LIN {X 0,Y 455.191,Z 1020.489,A -85,B 0,C 180,E1 17138.452,E2 17138.452} C_VEL
LIN {X 0,Y 455.669,Z 1006.442,A -85,B 0,C 180,E1 17140.566,E2 17140.566} C_VEL
LIN {X 0,Y 455.288,Z 999.068,A -85,B 0,C 180,E1 17142.573,E2 17142.573} C_VEL
LIN {X 0,Y 455.108,Z 997.219,A -85,B 0,C 180,E1 17144.205,E2 17144.205} C_VEL
LIN {X 0,Y 455.545,Z 998.35,A -85,B 0,C 180,E1 17145.874,E2 17145.874} C_VEL
LIN {X 0,Y 456.74,Z 1004.121,A -85,B 0,C 180,E1 17147.844,E2 17147.844} C_VEL
LIN {X 0,Y 457.689,Z 1016.104,A -85,B 0,C 180,E1 17149.82,E2 17149.82} C_VEL
LIN {X 0,Y 444.133,Z 1065.097,A -85,B 0,C 180,E1 17152.938,E2 17152.938} C_VEL
LIN {X 0,Y 432.896,Z 1103.693,A -85,B 0,C 180,E1 17156.355,E2 17156.355} C_VEL
LIN {X 0,Y 423.034,Z 1137.682,A -85,B 0,C 180,E1 17160.428,E2 17160.428} C_VEL
LIN {X 0,Y 415.2,Z 1166.581,A -85,B 0,C 180,E1 17165.098,E2 17165.098} C_VEL
LIN {X 0,Y 409.503,Z 1190.101,A -85,B 0,C 180,E1 17170.266,E2 17170.266} C_VEL
LIN {X 0,Y 406.234,Z 1207.399,A -85,B 0,C 180,E1 17175.641,E2 17175.641} C_VEL
LIN {X 0,Y 404.984,Z 1217.471,A -85,B 0,C 180,E1 17180.354,E2 17180.354} C_VEL
LIN {X 0,Y 404.678,Z 1223.746,A -85,B 0,C 180,E1 17185.736,E2 17185.736} C_VEL
LIN {X 0,Y 404.807,Z 1224.763,A -85,B 0,C 180,E1 17190.019,E2 17190.019} C_VEL
LIN {X 0,Y 404.778,Z 1222.047,A -85,B 0,C 180,E1 17194.3,E2 17194.3} C_VEL
LIN {X 0,Y 405.06,Z 1214.69,A -85,B 0,C 180,E1 17199.07,E2 17199.07} C_VEL
LIN {X 0,Y 406.066,Z 1201.006,A -85,B 0,C 180,E1 17204.275,E2 17204.275} C_VEL
LIN {X 0,Y 408.461,Z 1181.997,A -85,B 0,C 180,E1 17209.185,E2 17209.185} C_VEL
LIN {X 0,Y 412.41,Z 1157.442,A -85,B 0,C 180,E1 17213.787,E2 17213.787} C_VEL
LIN {X 0,Y 415.814,Z 1137.737,A -85,B 0,C 180,E1 17216.659,E2 17216.659} C_VEL
LIN {X 0,Y 414.066,Z 1125.291,A -85,B 0,C 180,E1 17218.355,E2 17218.355} C_VEL
LIN {X 0,Y 412.797,Z 1112.236,A -85,B 0,C 180,E1 17219.965,E2 17219.965} C_VEL
LIN {X 0,Y 419.177,Z 1075.451,A -85,B 0,C 180,E1 17223.278,E2 17223.278} C_VEL
LIN {X 0,Y 425.157,Z 1036.536,A -85,B 0,C 180,E1 17225.763,E2 17225.763} C_VEL
LIN {X 0,Y 427.532,Z 1011.003,A -85,B 0,C 180,E1 17226.997,E2 17226.997} C_VEL
LIN {X 0,Y 412.782,Z 969.477,A -85,B 0,C 180,E1 17229.572,E2 17229.572} C_VEL
LIN {X 0,Y 394.48,Z 923.03,A -85,B 0,C 180,E1 17232.402,E2 17232.402} C_VEL
LIN {X 0,Y 394.418,Z 923.03,A -85,B 0,C 180,E1 17239.363,E2 17239.363} C_VEL
LIN {X 0,Y 394.483,Z 923.03,A -85,B 0,C 180,E1 17244.932,E2 17244.932} C_VEL
LIN {X 0,Y 394.701,Z 923.03,A -85,B 0,C 180,E1 17251.739,E2 17251.739} C_VEL
LIN {X 0,Y 394.927,Z 923.03,A -85,B 0,C 180,E1 17257.506,E2 17257.506} C_VEL
LIN {X 0,Y 395.1,Z 923.497,A -85,B 0,C 180,E1 17261.03,E2 17261.03} C_VEL
LIN {X 0,Y 410.539,Z 954.287,A -85,B 0,C 180,E1 17264.343,E2 17264.343} C_VEL
LIN {X 0,Y 418.882,Z 977.95,A -85,B 0,C 180,E1 17266.049,E2 17266.049} C_VEL
LIN {X 0,Y 417.597,Z 1017.766,A -85,B 0,C 180,E1 17267.413,E2 17267.413} C_VEL
LIN {X 0,Y 415.215,Z 1045.588,A -85,B 0,C 180,E1 17269.12,E2 17269.12} C_VEL
LIN {X 0,Y 411.761,Z 1070.714,A -85,B 0,C 180,E1 17271.561,E2 17271.561} C_VEL
LIN {X 0,Y 407.999,Z 1092.019,A -85,B 0,C 180,E1 17274.69,E2 17274.69} C_VEL
LIN {X 0,Y 404.788,Z 1106.271,A -85,B 0,C 180,E1 17277.863,E2 17277.863} C_VEL
LIN {X 0,Y 401.89,Z 1116.644,A -85,B 0,C 180,E1 17281.618,E2 17281.618} C_VEL
LIN {X 0,Y 400.472,Z 1120.583,A -85,B 0,C 180,E1 17284.33,E2 17284.33} C_VEL
LIN {X 0,Y 399.572,Z 1121.825,A -85,B 0,C 180,E1 17286.517,E2 17286.517} C_VEL
LIN {X 0,Y 398.954,Z 1120.435,A -85,B 0,C 180,E1 17289.927,E2 17289.927} C_VEL
LIN {X 0,Y 398.958,Z 1113.006,A -85,B 0,C 180,E1 17294.154,E2 17294.154} C_VEL
LIN {X 0,Y 399.592,Z 1100.151,A -85,B 0,C 180,E1 17297.989,E2 17297.989} C_VEL
LIN {X 0,Y 400.849,Z 1081.362,A -85,B 0,C 180,E1 17301.567,E2 17301.567} C_VEL
LIN {X 0,Y 402.466,Z 1057.576,A -85,B 0,C 180,E1 17304.592,E2 17304.592} C_VEL
LIN {X 0,Y 404.027,Z 1030.386,A -85,B 0,C 180,E1 17306.89,E2 17306.89} C_VEL
LIN {X 0,Y 405.109,Z 1000.703,A -85,B 0,C 180,E1 17308.434,E2 17308.434} C_VEL
LIN {X 0,Y 404.88,Z 969.297,A -85,B 0,C 180,E1 17309.301,E2 17309.301} C_VEL
LIN {X 0,Y 394.897,Z 923.03,A -85,B 0,C 180,E1 17310.777,E2 17310.777} C_VEL
LIN {X 0,Y 394.426,Z 923.03,A -85,B 0,C 180,E1 17317.808,E2 17317.808} C_VEL
LIN {X 0,Y 394.391,Z 923.03,A -85,B 0,C 180,E1 17323.607,E2 17323.607} C_VEL
LIN {X 0,Y 394.447,Z 923.03,A -85,B 0,C 180,E1 17330.016,E2 17330.016} C_VEL
LIN {X 0,Y 394.553,Z 923.03,A -85,B 0,C 180,E1 17337.556,E2 17337.556} C_VEL
LIN {X 0,Y 394.819,Z 923.03,A -85,B 0,C 180,E1 17342.64,E2 17342.64} C_VEL
LIN {X 0,Y 395.179,Z 923.03,A -85,B 0,C 180,E1 17349.852,E2 17349.852} C_VEL
LIN {X 0,Y 395.545,Z 923.03,A -85,B 0,C 180,E1 17356.73,E2 17356.73} C_VEL
LIN {X 0,Y 396.026,Z 923.03,A -85,B 0,C 180,E1 17363.408,E2 17363.408} C_VEL
LIN {X 0,Y 396.58,Z 923.03,A -85,B 0,C 180,E1 17369.981,E2 17369.981} C_VEL
LIN {X 0,Y 395.971,Z 923.03,A -85,B 0,C 180,E1 17377.139,E2 17377.139} C_VEL
LIN {X 0,Y 395.625,Z 923.03,A -85,B 0,C 180,E1 17383.227,E2 17383.227} C_VEL
LIN {X 0,Y 395.195,Z 923.03,A -85,B 0,C 180,E1 17390.106,E2 17390.106} C_VEL
LIN {X 0,Y 394.82,Z 923.03,A -85,B 0,C 180,E1 17397.316,E2 17397.316} C_VEL
LIN {X 0,Y 394.598,Z 923.03,A -85,B 0,C 180,E1 17402.593,E2 17402.593} C_VEL
LIN {X 0,Y 394.468,Z 923.03,A -85,B 0,C 180,E1 17409.988,E2 17409.988} C_VEL
LIN {X 0,Y 394.457,Z 923.03,A -85,B 0,C 180,E1 17416.673,E2 17416.673} C_VEL
LIN {X 0,Y 394.548,Z 923.058,A -85,B 0,C 180,E1 17418.728,E2 17418.728} C_VEL
LIN {X 0,Y 410.897,Z 967.63,A -85,B 0,C 180,E1 17421.625,E2 17421.625} C_VEL
LIN {X 0,Y 422.679,Z 1006.495,A -85,B 0,C 180,E1 17424.633,E2 17424.633} C_VEL
LIN {X 0,Y 424.124,Z 1014.104,A -85,B 0,C 180,E1 17425.243,E2 17425.243} C_VEL
LIN {X 0,Y 417.97,Z 1053.429,A -85,B 0,C 180,E1 17428.199,E2 17428.199} C_VEL
LIN {X 0,Y 412.029,Z 1087.161,A -85,B 0,C 180,E1 17431.706,E2 17431.706} C_VEL
LIN {X 0,Y 406.484,Z 1116.868,A -85,B 0,C 180,E1 17435.86,E2 17435.86} C_VEL
LIN {X 0,Y 402.138,Z 1141.556,A -85,B 0,C 180,E1 17440.517,E2 17440.517} C_VEL
LIN {X 0,Y 399.018,Z 1161.589,A -85,B 0,C 180,E1 17445.747,E2 17445.747} C_VEL
LIN {X 0,Y 397.442,Z 1175.743,A -85,B 0,C 180,E1 17451.25,E2 17451.25} C_VEL
LIN {X 0,Y 396.827,Z 1183.919,A -85,B 0,C 180,E1 17456.723,E2 17456.723} C_VEL
LIN {X 0,Y 396.94,Z 1186.66,A -85,B 0,C 180,E1 17462.179,E2 17462.179} C_VEL
LIN {X 0,Y 397.795,Z 1184.171,A -85,B 0,C 180,E1 17467.638,E2 17467.638} C_VEL
LIN {X 0,Y 399.762,Z 1176.484,A -85,B 0,C 180,E1 17473.106,E2 17473.106} C_VEL
LIN {X 0,Y 403.759,Z 1163.247,A -85,B 0,C 180,E1 17478.547,E2 17478.547} C_VEL
LIN {X 0,Y 410.22,Z 1143.839,A -85,B 0,C 180,E1 17483.901,E2 17483.901} C_VEL
LIN {X 0,Y 419.067,Z 1118.652,A -85,B 0,C 180,E1 17488.832,E2 17488.832} C_VEL
LIN {X 0,Y 429.475,Z 1088.982,A -85,B 0,C 180,E1 17493.047,E2 17493.047} C_VEL
LIN {X 0,Y 442.014,Z 1052.06,A -85,B 0,C 180,E1 17496.896,E2 17496.896} C_VEL
LIN {X 0,Y 450.785,Z 1024.289,A -85,B 0,C 180,E1 17499.132,E2 17499.132} C_VEL
LIN {X 0,Y 451.859,Z 1011.926,A -85,B 0,C 180,E1 17501.112,E2 17501.112} C_VEL
LIN {X 0,Y 452.025,Z 1006.374,A -85,B 0,C 180,E1 17502.686,E2 17502.686} C_VEL
LIN {X 0,Y 452.023,Z 1004.71,A -85,B 0,C 180,E1 17504.587,E2 17504.587} C_VEL
LIN {X 0,Y 452.818,Z 1007.731,A -85,B 0,C 180,E1 17506.73,E2 17506.73} C_VEL
LIN {X 0,Y 453.398,Z 1017.576,A -85,B 0,C 180,E1 17508.786,E2 17508.786} C_VEL
LIN {X 0,Y 452.878,Z 1022.13,A -85,B 0,C 180,E1 17509.304,E2 17509.304} C_VEL
LIN {X 0,Y 439.917,Z 1063.67,A -85,B 0,C 180,E1 17511.957,E2 17511.957} C_VEL
LIN {X 0,Y 427.232,Z 1103.723,A -85,B 0,C 180,E1 17515.56,E2 17515.56} C_VEL
LIN {X 0,Y 416.484,Z 1138.178,A -85,B 0,C 180,E1 17519.798,E2 17519.798} C_VEL
LIN {X 0,Y 408.15,Z 1166.565,A -85,B 0,C 180,E1 17524.506,E2 17524.506} C_VEL
LIN {X 0,Y 402.053,Z 1189.788,A -85,B 0,C 180,E1 17529.736,E2 17529.736} C_VEL
LIN {X 0,Y 398.415,Z 1207.747,A -85,B 0,C 180,E1 17535.518,E2 17535.518} C_VEL
LIN {X 0,Y 397.016,Z 1218.96,A -85,B 0,C 180,E1 17541.263,E2 17541.263} C_VEL
LIN {X 0,Y 396.773,Z 1223.391,A -85,B 0,C 180,E1 17545.651,E2 17545.651} C_VEL
LIN {X 0,Y 396.918,Z 1224.311,A -85,B 0,C 180,E1 17550.019,E2 17550.019} C_VEL
LIN {X 0,Y 396.969,Z 1220.195,A -85,B 0,C 180,E1 17555.48,E2 17555.48} C_VEL
LIN {X 0,Y 397.36,Z 1210.042,A -85,B 0,C 180,E1 17560.98,E2 17560.98} C_VEL
LIN {X 0,Y 398.92,Z 1194.207,A -85,B 0,C 180,E1 17566.241,E2 17566.241} C_VEL
LIN {X 0,Y 402.034,Z 1172.688,A -85,B 0,C 180,E1 17571.227,E2 17571.227} C_VEL
LIN {X 0,Y 406.523,Z 1146.891,A -85,B 0,C 180,E1 17575.62,E2 17575.62} C_VEL
LIN {X 0,Y 412.088,Z 1116.105,A -85,B 0,C 180,E1 17579.539,E2 17579.539} C_VEL
LIN {X 0,Y 412.797,Z 1112.236,A -85,B 0,C 180,E1 17579.965,E2 17579.965} C_VEL
LIN {X 0,Y 411.653,Z 1098.605,A -85,B 0,C 180,E1 17581.486,E2 17581.486} C_VEL
LIN {X 0,Y 410.27,Z 1084.427,A -85,B 0,C 180,E1 17582.924,E2 17582.924} C_VEL
LIN {X 0,Y 416.384,Z 1046.661,A -85,B 0,C 180,E1 17585.619,E2 17585.619} C_VEL
LIN {X 0,Y 420.389,Z 1013.535,A -85,B 0,C 180,E1 17587.322,E2 17587.322} C_VEL
LIN {X 0,Y 406.01,Z 972.479,A -85,B 0,C 180,E1 17589.966,E2 17589.966} C_VEL
LIN {X 0,Y 386.525,Z 923.03,A -85,B 0,C 180,E1 17593.043,E2 17593.043} C_VEL
LIN {X 0,Y 386.41,Z 923.03,A -85,B 0,C 180,E1 17598.336,E2 17598.336} C_VEL
LIN {X 0,Y 386.579,Z 923.03,A -85,B 0,C 180,E1 17605.199,E2 17605.199} C_VEL
LIN {X 0,Y 386.829,Z 923.03,A -85,B 0,C 180,E1 17612.049,E2 17612.049} C_VEL
LIN {X 0,Y 387.149,Z 923.418,A -85,B 0,C 180,E1 17619.685,E2 17619.685} C_VEL
LIN {X 0,Y 390.017,Z 929.079,A -85,B 0,C 180,E1 17620.451,E2 17620.451} C_VEL
LIN {X 0,Y 403.178,Z 954.398,A -85,B 0,C 180,E1 17623.437,E2 17623.437} C_VEL
LIN {X 0,Y 412.347,Z 979.36,A -85,B 0,C 180,E1 17625.406,E2 17625.406} C_VEL
LIN {X 0,Y 411.141,Z 1018.392,A -85,B 0,C 180,E1 17626.79,E2 17626.79} C_VEL
LIN {X 0,Y 408.388,Z 1048.042,A -85,B 0,C 180,E1 17628.666,E2 17628.666} C_VEL
LIN {X 0,Y 404.74,Z 1072.75,A -85,B 0,C 180,E1 17631.143,E2 17631.143} C_VEL
LIN {X 0,Y 400.748,Z 1093.641,A -85,B 0,C 180,E1 17634.322,E2 17634.322} C_VEL
LIN {X 0,Y 397.096,Z 1108.65,A -85,B 0,C 180,E1 17637.821,E2 17637.821} C_VEL
LIN {X 0,Y 394.413,Z 1117.39,A -85,B 0,C 180,E1 17641.1,E2 17641.1} C_VEL
LIN {X 0,Y 392.608,Z 1121.967,A -85,B 0,C 180,E1 17644.417,E2 17644.417} C_VEL
LIN {X 0,Y 391.706,Z 1122.946,A -85,B 0,C 180,E1 17646.648,E2 17646.648} C_VEL
LIN {X 0,Y 391.083,Z 1121.036,A -85,B 0,C 180,E1 17650.129,E2 17650.129} C_VEL
LIN {X 0,Y 391.148,Z 1112.544,A -85,B 0,C 180,E1 17654.61,E2 17654.61} C_VEL
LIN {X 0,Y 391.797,Z 1099.582,A -85,B 0,C 180,E1 17658.321,E2 17658.321} C_VEL
LIN {X 0,Y 393.034,Z 1081.576,A -85,B 0,C 180,E1 17661.721,E2 17661.721} C_VEL
LIN {X 0,Y 394.668,Z 1057.76,A -85,B 0,C 180,E1 17664.766,E2 17664.766} C_VEL
LIN {X 0,Y 396.301,Z 1029.898,A -85,B 0,C 180,E1 17667.129,E2 17667.129} C_VEL
LIN {X 0,Y 397.389,Z 1000.153,A -85,B 0,C 180,E1 17668.672,E2 17668.672} C_VEL
LIN {X 0,Y 397.135,Z 970.302,A -85,B 0,C 180,E1 17669.506,E2 17669.506} C_VEL
LIN {X 0,Y 386.973,Z 923.03,A -85,B 0,C 180,E1 17671,E2 17671} C_VEL
LIN {X 0,Y 386.453,Z 923.03,A -85,B 0,C 180,E1 17678.731,E2 17678.731} C_VEL
LIN {X 0,Y 386.383,Z 923.03,A -85,B 0,C 180,E1 17685.232,E2 17685.232} C_VEL
LIN {X 0,Y 386.494,Z 923.03,A -85,B 0,C 180,E1 17691.443,E2 17691.443} C_VEL
LIN {X 0,Y 386.585,Z 923.03,A -85,B 0,C 180,E1 17696.802,E2 17696.802} C_VEL
LIN {X 0,Y 386.907,Z 923.03,A -85,B 0,C 180,E1 17703.939,E2 17703.939} C_VEL
LIN {X 0,Y 387.224,Z 923.03,A -85,B 0,C 180,E1 17709.491,E2 17709.491} C_VEL
LIN {X 0,Y 387.629,Z 923.03,A -85,B 0,C 180,E1 17717.063,E2 17717.063} C_VEL
LIN {X 0,Y 388.119,Z 923.03,A -85,B 0,C 180,E1 17723.273,E2 17723.273} C_VEL
LIN {X 0,Y 388.677,Z 923.03,A -85,B 0,C 180,E1 17729.98,E2 17729.98} C_VEL
LIN {X 0,Y 388.146,Z 923.03,A -85,B 0,C 180,E1 17736.687,E2 17736.687} C_VEL
LIN {X 0,Y 387.682,Z 923.03,A -85,B 0,C 180,E1 17743.503,E2 17743.503} C_VEL
LIN {X 0,Y 387.225,Z 923.03,A -85,B 0,C 180,E1 17750.539,E2 17750.539} C_VEL
LIN {X 0,Y 386.881,Z 923.03,A -85,B 0,C 180,E1 17757.925,E2 17757.925} C_VEL
LIN {X 0,Y 386.571,Z 923.03,A -85,B 0,C 180,E1 17765.87,E2 17765.87} C_VEL
LIN {X 0,Y 386.451,Z 923.03,A -85,B 0,C 180,E1 17772.014,E2 17772.014} C_VEL
LIN {X 0,Y 386.608,Z 923.177,A -85,B 0,C 180,E1 17778.099,E2 17778.099} C_VEL
LIN {X 0,Y 403.089,Z 967.84,A -85,B 0,C 180,E1 17781.079,E2 17781.079} C_VEL
LIN {X 0,Y 415.016,Z 1007.284,A -85,B 0,C 180,E1 17784.201,E2 17784.201} C_VEL
LIN {X 0,Y 416.619,Z 1016.141,A -85,B 0,C 180,E1 17784.925,E2 17784.925} C_VEL
LIN {X 0,Y 410.408,Z 1054.702,A -85,B 0,C 180,E1 17787.91,E2 17787.91} C_VEL
LIN {X 0,Y 404.319,Z 1088.358,A -85,B 0,C 180,E1 17791.492,E2 17791.492} C_VEL
LIN {X 0,Y 398.749,Z 1117.52,A -85,B 0,C 180,E1 17795.659,E2 17795.659} C_VEL
LIN {X 0,Y 394.092,Z 1143.431,A -85,B 0,C 180,E1 17800.685,E2 17800.685} C_VEL
LIN {X 0,Y 390.972,Z 1163.224,A -85,B 0,C 180,E1 17806.095,E2 17806.095} C_VEL
LIN {X 0,Y 389.616,Z 1175.758,A -85,B 0,C 180,E1 17811.073,E2 17811.073} C_VEL
LIN {X 0,Y 388.933,Z 1184.165,A -85,B 0,C 180,E1 17816.657,E2 17816.657} C_VEL
LIN {X 0,Y 389.052,Z 1187.126,A -85,B 0,C 180,E1 17822.224,E2 17822.224} C_VEL
LIN {X 0,Y 389.716,Z 1185.689,A -85,B 0,C 180,E1 17826.678,E2 17826.678} C_VEL
LIN {X 0,Y 391.543,Z 1179.288,A -85,B 0,C 180,E1 17832.253,E2 17832.253} C_VEL
LIN {X 0,Y 395.288,Z 1167.515,A -85,B 0,C 180,E1 17837.805,E2 17837.805} C_VEL
LIN {X 0,Y 401.929,Z 1148.838,A -85,B 0,C 180,E1 17843.542,E2 17843.542} C_VEL
LIN {X 0,Y 410.81,Z 1125.289,A -85,B 0,C 180,E1 17848.564,E2 17848.564} C_VEL
LIN {X 0,Y 421.943,Z 1095.977,A -85,B 0,C 180,E1 17853.1,E2 17853.1} C_VEL
LIN {X 0,Y 435.131,Z 1060.593,A -85,B 0,C 180,E1 17857.089,E2 17857.089} C_VEL
LIN {X 0,Y 446.809,Z 1027.128,A -85,B 0,C 180,E1 17859.981,E2 17859.981} C_VEL
LIN {X 0,Y 448.315,Z 1016.57,A -85,B 0,C 180,E1 17861.881,E2 17861.881} C_VEL
LIN {X 0,Y 448.619,Z 1013.196,A -85,B 0,C 180,E1 17863.088,E2 17863.088} C_VEL
LIN {X 0,Y 448.961,Z 1012.29,A -85,B 0,C 180,E1 17865.053,E2 17865.053} C_VEL
LIN {X 0,Y 449.458,Z 1015.621,A -85,B 0,C 180,E1 17866.789,E2 17866.789} C_VEL
LIN {X 0,Y 449.249,Z 1023.398,A -85,B 0,C 180,E1 17868.339,E2 17868.339} C_VEL
LIN {X 0,Y 432.879,Z 1071.725,A -85,B 0,C 180,E1 17871.686,E2 17871.686} C_VEL
LIN {X 0,Y 419.59,Z 1110.488,A -85,B 0,C 180,E1 17875.47,E2 17875.47} C_VEL
LIN {X 0,Y 408.639,Z 1143.005,A -85,B 0,C 180,E1 17879.771,E2 17879.771} C_VEL
LIN {X 0,Y 399.672,Z 1171.598,A -85,B 0,C 180,E1 17884.911,E2 17884.911} C_VEL
LIN {X 0,Y 394.089,Z 1191.813,A -85,B 0,C 180,E1 17889.835,E2 17889.835} C_VEL
LIN {X 0,Y 390.661,Z 1207.717,A -85,B 0,C 180,E1 17895.233,E2 17895.233} C_VEL
LIN {X 0,Y 389.284,Z 1217.092,A -85,B 0,C 180,E1 17899.961,E2 17899.961} C_VEL
LIN {X 0,Y 388.882,Z 1223.045,A -85,B 0,C 180,E1 17905.563,E2 17905.563} C_VEL
LIN {X 0,Y 389.032,Z 1223.821,A -85,B 0,C 180,E1 17910.02,E2 17910.02} C_VEL
LIN {X 0,Y 389.1,Z 1219.525,A -85,B 0,C 180,E1 17915.591,E2 17915.591} C_VEL
LIN {X 0,Y 389.439,Z 1210.457,A -85,B 0,C 180,E1 17920.64,E2 17920.64} C_VEL
LIN {X 0,Y 390.765,Z 1195.999,A -85,B 0,C 180,E1 17925.724,E2 17925.724} C_VEL
LIN {X 0,Y 393.948,Z 1174.002,A -85,B 0,C 180,E1 17931.095,E2 17931.095} C_VEL
LIN {X 0,Y 398.793,Z 1146.835,A -85,B 0,C 180,E1 17935.852,E2 17935.852} C_VEL
LIN {X 0,Y 404.49,Z 1116.115,A -85,B 0,C 180,E1 17939.842,E2 17939.842} C_VEL
LIN {X 0,Y 410.27,Z 1084.427,A -85,B 0,C 180,E1 17942.924,E2 17942.924} C_VEL
LIN {X 0,Y 408.992,Z 1069.918,A -85,B 0,C 180,E1 17944.271,E2 17944.271} C_VEL
LIN {X 0,Y 407.83,Z 1054.806,A -85,B 0,C 180,E1 17945.533,E2 17945.533} C_VEL
LIN {X 0,Y 412.988,Z 1015.191,A -85,B 0,C 180,E1 17947.709,E2 17947.709} C_VEL
LIN {X 0,Y 398.465,Z 973.55,A -85,B 0,C 180,E1 17950.479,E2 17950.479} C_VEL
LIN {X 0,Y 378.612,Z 923.03,A -85,B 0,C 180,E1 17953.698,E2 17953.698} C_VEL
LIN {X 0,Y 378.45,Z 923.03,A -85,B 0,C 180,E1 17960.296,E2 17960.296} C_VEL
LIN {X 0,Y 378.694,Z 923.03,A -85,B 0,C 180,E1 17966.954,E2 17966.954} C_VEL
LIN {X 0,Y 378.953,Z 923.03,A -85,B 0,C 180,E1 17973.986,E2 17973.986} C_VEL
LIN {X 0,Y 379.063,Z 923.637,A -85,B 0,C 180,E1 17978.14,E2 17978.14} C_VEL
LIN {X 0,Y 382.013,Z 929.148,A -85,B 0,C 180,E1 17979.015,E2 17979.015} C_VEL
LIN {X 0,Y 394.22,Z 951.156,A -85,B 0,C 180,E1 17982.065,E2 17982.065} C_VEL
LIN {X 0,Y 404.2,Z 975.224,A -85,B 0,C 180,E1 17984.325,E2 17984.325} C_VEL
LIN {X 0,Y 406.502,Z 984.421,A -85,B 0,C 180,E1 17984.92,E2 17984.92} C_VEL
LIN {X 0,Y 404.697,Z 1020.079,A -85,B 0,C 180,E1 17986.19,E2 17986.19} C_VEL
LIN {X 0,Y 401.963,Z 1047.836,A -85,B 0,C 180,E1 17987.96,E2 17987.96} C_VEL
LIN {X 0,Y 398.122,Z 1072.669,A -85,B 0,C 180,E1 17990.444,E2 17990.444} C_VEL
LIN {X 0,Y 393.828,Z 1093.968,A -85,B 0,C 180,E1 17993.669,E2 17993.669} C_VEL
LIN {X 0,Y 389.879,Z 1109.217,A -85,B 0,C 180,E1 17997.225,E2 17997.225} C_VEL
LIN {X 0,Y 386.636,Z 1119.204,A -85,B 0,C 180,E1 18001.122,E2 18001.122} C_VEL
LIN {X 0,Y 384.754,Z 1123.332,A -85,B 0,C 180,E1 18004.508,E2 18004.508} C_VEL
LIN {X 0,Y 383.831,Z 1123.953,A -85,B 0,C 180,E1 18006.785,E2 18006.785} C_VEL
LIN {X 0,Y 383.217,Z 1121.694,A -85,B 0,C 180,E1 18010.274,E2 18010.274} C_VEL
LIN {X 0,Y 383.241,Z 1113.809,A -85,B 0,C 180,E1 18014.407,E2 18014.407} C_VEL
LIN {X 0,Y 383.926,Z 1100.316,A -85,B 0,C 180,E1 18018.356,E2 18018.356} C_VEL
LIN {X 0,Y 385.219,Z 1081.747,A -85,B 0,C 180,E1 18021.882,E2 18021.882} C_VEL
LIN {X 0,Y 386.903,Z 1057.619,A -85,B 0,C 180,E1 18024.982,E2 18024.982} C_VEL
LIN {X 0,Y 388.555,Z 1029.791,A -85,B 0,C 180,E1 18027.344,E2 18027.344} C_VEL
LIN {X 0,Y 389.674,Z 999.259,A -85,B 0,C 180,E1 18028.914,E2 18028.914} C_VEL
LIN {X 0,Y 389.293,Z 971.002,A -85,B 0,C 180,E1 18029.716,E2 18029.716} C_VEL
LIN {X 0,Y 379.01,Z 923.03,A -85,B 0,C 180,E1 18031.312,E2 18031.312} C_VEL
LIN {X 0,Y 378.419,Z 923.03,A -85,B 0,C 180,E1 18039.714,E2 18039.714} C_VEL
LIN {X 0,Y 378.425,Z 923.03,A -85,B 0,C 180,E1 18047.225,E2 18047.225} C_VEL
LIN {X 0,Y 378.515,Z 923.03,A -85,B 0,C 180,E1 18053.193,E2 18053.193} C_VEL
LIN {X 0,Y 378.715,Z 923.03,A -85,B 0,C 180,E1 18058.734,E2 18058.734} C_VEL
LIN {X 0,Y 379.024,Z 923.03,A -85,B 0,C 180,E1 18063.969,E2 18063.969} C_VEL
LIN {X 0,Y 379.37,Z 923.03,A -85,B 0,C 180,E1 18071.399,E2 18071.399} C_VEL
LIN {X 0,Y 379.807,Z 923.03,A -85,B 0,C 180,E1 18078.506,E2 18078.506} C_VEL
LIN {X 0,Y 380.386,Z 923.03,A -85,B 0,C 180,E1 18085.423,E2 18085.423} C_VEL
LIN {X 0,Y 380.774,Z 923.03,A -85,B 0,C 180,E1 18089.98,E2 18089.98} C_VEL
LIN {X 0,Y 380.223,Z 923.03,A -85,B 0,C 180,E1 18096.827,E2 18096.827} C_VEL
LIN {X 0,Y 379.729,Z 923.03,A -85,B 0,C 180,E1 18103.792,E2 18103.792} C_VEL
LIN {X 0,Y 379.241,Z 923.03,A -85,B 0,C 180,E1 18110.991,E2 18110.991} C_VEL
LIN {X 0,Y 378.886,Z 923.03,A -85,B 0,C 180,E1 18118.663,E2 18118.663} C_VEL
LIN {X 0,Y 378.71,Z 923.03,A -85,B 0,C 180,E1 18123.932,E2 18123.932} C_VEL
LIN {X 0,Y 378.489,Z 923.03,A -85,B 0,C 180,E1 18130.658,E2 18130.658} C_VEL
LIN {X 0,Y 378.607,Z 923.253,A -85,B 0,C 180,E1 18137.439,E2 18137.439} C_VEL
LIN {X 0,Y 395.119,Z 967.893,A -85,B 0,C 180,E1 18140.502,E2 18140.502} C_VEL
LIN {X 0,Y 407.37,Z 1008.192,A -85,B 0,C 180,E1 18143.776,E2 18143.776} C_VEL
LIN {X 0,Y 409.045,Z 1018.506,A -85,B 0,C 180,E1 18144.636,E2 18144.636} C_VEL
LIN {X 0,Y 402.868,Z 1055.772,A -85,B 0,C 180,E1 18147.599,E2 18147.599} C_VEL
LIN {X 0,Y 396.693,Z 1089.099,A -85,B 0,C 180,E1 18151.221,E2 18151.221} C_VEL
LIN {X 0,Y 390.713,Z 1119.827,A -85,B 0,C 180,E1 18155.734,E2 18155.734} C_VEL
LIN {X 0,Y 386.046,Z 1145.21,A -85,B 0,C 180,E1 18160.869,E2 18160.869} C_VEL
LIN {X 0,Y 383.166,Z 1163.089,A -85,B 0,C 180,E1 18165.857,E2 18165.857} C_VEL
LIN {X 0,Y 381.77,Z 1175.747,A -85,B 0,C 180,E1 18170.888,E2 18170.888} C_VEL
LIN {X 0,Y 381.04,Z 1184.401,A -85,B 0,C 180,E1 18176.587,E2 18176.587} C_VEL
LIN {X 0,Y 381.165,Z 1187.594,A -85,B 0,C 180,E1 18182.27,E2 18182.27} C_VEL
LIN {X 0,Y 381.886,Z 1186.318,A -85,B 0,C 180,E1 18186.815,E2 18186.815} C_VEL
LIN {X 0,Y 383.838,Z 1180.174,A -85,B 0,C 180,E1 18192.502,E2 18192.502} C_VEL
LIN {X 0,Y 387.84,Z 1168.714,A -85,B 0,C 180,E1 18198.159,E2 18198.159} C_VEL
LIN {X 0,Y 394.407,Z 1151.476,A -85,B 0,C 180,E1 18203.717,E2 18203.717} C_VEL
LIN {X 0,Y 404.2,Z 1127.63,A -85,B 0,C 180,E1 18209.076,E2 18209.076} C_VEL
LIN {X 0,Y 416.587,Z 1097.444,A -85,B 0,C 180,E1 18213.894,E2 18213.894} C_VEL
LIN {X 0,Y 430.972,Z 1062.064,A -85,B 0,C 180,E1 18217.978,E2 18217.978} C_VEL
LIN {X 0,Y 442.694,Z 1032.353,A -85,B 0,C 180,E1 18220.539,E2 18220.539} C_VEL
LIN {X 0,Y 444.745,Z 1022.854,A -85,B 0,C 180,E1 18222.295,E2 18222.295} C_VEL
LIN {X 0,Y 445.053,Z 1021.301,A -85,B 0,C 180,E1 18222.768,E2 18222.768} C_VEL
LIN {X 0,Y 445.399,Z 1019.471,A -85,B 0,C 180,E1 18224.594,E2 18224.594} C_VEL
LIN {X 0,Y 445.828,Z 1021.012,A -85,B 0,C 180,E1 18226.072,E2 18226.072} C_VEL
LIN {X 0,Y 445.33,Z 1027.959,A -85,B 0,C 180,E1 18227.669,E2 18227.669} C_VEL
LIN {X 0,Y 429.521,Z 1069.82,A -85,B 0,C 180,E1 18230.574,E2 18230.574} C_VEL
LIN {X 0,Y 414.912,Z 1108.73,A -85,B 0,C 180,E1 18234.385,E2 18234.385} C_VEL
LIN {X 0,Y 402.513,Z 1142.706,A -85,B 0,C 180,E1 18238.948,E2 18238.948} C_VEL
LIN {X 0,Y 393.021,Z 1170.744,A -85,B 0,C 180,E1 18244.089,E2 18244.089} C_VEL
LIN {X 0,Y 386.563,Z 1192.091,A -85,B 0,C 180,E1 18249.425,E2 18249.425} C_VEL
LIN {X 0,Y 382.88,Z 1207.71,A -85,B 0,C 180,E1 18254.926,E2 18254.926} C_VEL
LIN {X 0,Y 381.411,Z 1216.933,A -85,B 0,C 180,E1 18259.751,E2 18259.751} C_VEL
LIN {X 0,Y 380.978,Z 1222.702,A -85,B 0,C 180,E1 18265.471,E2 18265.471} C_VEL
LIN {X 0,Y 381.147,Z 1223.296,A -85,B 0,C 180,E1 18270.02,E2 18270.02} C_VEL
LIN {X 0,Y 381.225,Z 1218.81,A -85,B 0,C 180,E1 18275.707,E2 18275.707} C_VEL
LIN {X 0,Y 381.581,Z 1209.582,A -85,B 0,C 180,E1 18280.862,E2 18280.862} C_VEL
LIN {X 0,Y 383.177,Z 1193.883,A -85,B 0,C 180,E1 18286.338,E2 18286.338} C_VEL
LIN {X 0,Y 386.392,Z 1172.445,A -85,B 0,C 180,E1 18291.527,E2 18291.527} C_VEL
LIN {X 0,Y 391.087,Z 1146.73,A -85,B 0,C 180,E1 18296.092,E2 18296.092} C_VEL
LIN {X 0,Y 396.894,Z 1116.042,A -85,B 0,C 180,E1 18300.157,E2 18300.157} C_VEL
LIN {X 0,Y 403.386,Z 1081.275,A -85,B 0,C 180,E1 18303.561,E2 18303.561} C_VEL
LIN {X 0,Y 407.83,Z 1054.806,A -85,B 0,C 180,E1 18305.533,E2 18305.533} C_VEL
LIN {X 0,Y 406.677,Z 1039.372,A -85,B 0,C 180,E1 18306.694,E2 18306.694} C_VEL
LIN {X 0,Y 405.245,Z 1023.527,A -85,B 0,C 180,E1 18307.743,E2 18307.743} C_VEL
LIN {X 0,Y 405.117,Z 1015.102,A -85,B 0,C 180,E1 18308.224,E2 18308.224} C_VEL
LIN {X 0,Y 390.195,Z 972.493,A -85,B 0,C 180,E1 18311.132,E2 18311.132} C_VEL
LIN {X 0,Y 370.613,Z 923.03,A -85,B 0,C 180,E1 18314.385,E2 18314.385} C_VEL
LIN {X 0,Y 370.519,Z 923.03,A -85,B 0,C 180,E1 18322.287,E2 18322.287} C_VEL
LIN {X 0,Y 370.801,Z 923.03,A -85,B 0,C 180,E1 18328.879,E2 18328.879} C_VEL
LIN {X 0,Y 371.103,Z 923.295,A -85,B 0,C 180,E1 18336.336,E2 18336.336} C_VEL
LIN {X 0,Y 373.684,Z 928.831,A -85,B 0,C 180,E1 18337.272,E2 18337.272} C_VEL
LIN {X 0,Y 383.739,Z 945.345,A -85,B 0,C 180,E1 18340.127,E2 18340.127} C_VEL
LIN {X 0,Y 394.853,Z 968.703,A -85,B 0,C 180,E1 18342.864,E2 18342.864} C_VEL
LIN {X 0,Y 400.37,Z 986.047,A -85,B 0,C 180,E1 18344.245,E2 18344.245} C_VEL
LIN {X 0,Y 398.413,Z 1021.249,A -85,B 0,C 180,E1 18345.534,E2 18345.534} C_VEL
LIN {X 0,Y 395.282,Z 1050.433,A -85,B 0,C 180,E1 18347.455,E2 18347.455} C_VEL
LIN {X 0,Y 391.204,Z 1074.867,A -85,B 0,C 180,E1 18349.992,E2 18349.992} C_VEL
LIN {X 0,Y 386.643,Z 1095.773,A -85,B 0,C 180,E1 18353.269,E2 18353.269} C_VEL
LIN {X 0,Y 382.739,Z 1109.854,A -85,B 0,C 180,E1 18356.607,E2 18356.607} C_VEL
LIN {X 0,Y 379.227,Z 1119.985,A -85,B 0,C 180,E1 18360.558,E2 18360.558} C_VEL
LIN {X 0,Y 376.878,Z 1124.614,A -85,B 0,C 180,E1 18364.602,E2 18364.602} C_VEL
LIN {X 0,Y 375.951,Z 1124.946,A -85,B 0,C 180,E1 18366.928,E2 18366.928} C_VEL
LIN {X 0,Y 375.339,Z 1122.238,A -85,B 0,C 180,E1 18370.44,E2 18370.44} C_VEL
LIN {X 0,Y 375.47,Z 1113.039,A -85,B 0,C 180,E1 18374.949,E2 18374.949} C_VEL
LIN {X 0,Y 376.247,Z 1098.406,A -85,B 0,C 180,E1 18378.973,E2 18378.973} C_VEL
LIN {X 0,Y 377.66,Z 1078.303,A -85,B 0,C 180,E1 18382.6,E2 18382.6} C_VEL
LIN {X 0,Y 379.401,Z 1052.882,A -85,B 0,C 180,E1 18385.669,E2 18385.669} C_VEL
LIN {X 0,Y 381.051,Z 1024.434,A -85,B 0,C 180,E1 18387.906,E2 18387.906} C_VEL
LIN {X 0,Y 382.008,Z 993.537,A -85,B 0,C 180,E1 18389.33,E2 18389.33} C_VEL
LIN {X 0,Y 381.433,Z 971.443,A -85,B 0,C 180,E1 18389.936,E2 18389.936} C_VEL
LIN {X 0,Y 371.066,Z 923.03,A -85,B 0,C 180,E1 18391.643,E2 18391.643} C_VEL
LIN {X 0,Y 370.467,Z 923.03,A -85,B 0,C 180,E1 18399.17,E2 18399.17} C_VEL
LIN {X 0,Y 370.51,Z 923.03,A -85,B 0,C 180,E1 18406.082,E2 18406.082} C_VEL
LIN {X 0,Y 370.515,Z 923.03,A -85,B 0,C 180,E1 18412.262,E2 18412.262} C_VEL
LIN {X 0,Y 370.812,Z 923.03,A -85,B 0,C 180,E1 18418.85,E2 18418.85} C_VEL
LIN {X 0,Y 371.135,Z 923.03,A -85,B 0,C 180,E1 18425.954,E2 18425.954} C_VEL
LIN {X 0,Y 371.568,Z 923.03,A -85,B 0,C 180,E1 18433.441,E2 18433.441} C_VEL
LIN {X 0,Y 372.063,Z 923.03,A -85,B 0,C 180,E1 18440.631,E2 18440.631} C_VEL
LIN {X 0,Y 372.71,Z 923.03,A -85,B 0,C 180,E1 18447.656,E2 18447.656} C_VEL
LIN {X 0,Y 372.702,Z 923.03,A -85,B 0,C 180,E1 18452.303,E2 18452.303} C_VEL
LIN {X 0,Y 372.094,Z 923.03,A -85,B 0,C 180,E1 18459.327,E2 18459.327} C_VEL
LIN {X 0,Y 371.635,Z 923.03,A -85,B 0,C 180,E1 18466.513,E2 18466.513} C_VEL
LIN {X 0,Y 371.143,Z 923.03,A -85,B 0,C 180,E1 18474.001,E2 18474.001} C_VEL
LIN {X 0,Y 370.856,Z 923.03,A -85,B 0,C 180,E1 18481.161,E2 18481.161} C_VEL
LIN {X 0,Y 370.551,Z 923.03,A -85,B 0,C 180,E1 18487.682,E2 18487.682} C_VEL
LIN {X 0,Y 370.561,Z 923.03,A -85,B 0,C 180,E1 18493.853,E2 18493.853} C_VEL
LIN {X 0,Y 370.637,Z 923.03,A -85,B 0,C 180,E1 18496.744,E2 18496.744} C_VEL
LIN {X 0,Y 387.321,Z 968.02,A -85,B 0,C 180,E1 18499.928,E2 18499.928} C_VEL
LIN {X 0,Y 399.187,Z 1007.102,A -85,B 0,C 180,E1 18503.157,E2 18503.157} C_VEL
LIN {X 0,Y 401.734,Z 1019.122,A -85,B 0,C 180,E1 18504.22,E2 18504.22} C_VEL
LIN {X 0,Y 395.355,Z 1056.72,A -85,B 0,C 180,E1 18507.27,E2 18507.27} C_VEL
LIN {X 0,Y 388.974,Z 1090.278,A -85,B 0,C 180,E1 18511.001,E2 18511.001} C_VEL
LIN {X 0,Y 382.945,Z 1120.522,A -85,B 0,C 180,E1 18515.545,E2 18515.545} C_VEL
LIN {X 0,Y 378.163,Z 1145.92,A -85,B 0,C 180,E1 18520.801,E2 18520.801} C_VEL
LIN {X 0,Y 375.202,Z 1164.087,A -85,B 0,C 180,E1 18526.014,E2 18526.014} C_VEL
LIN {X 0,Y 373.71,Z 1177.299,A -85,B 0,C 180,E1 18531.553,E2 18531.553} C_VEL
LIN {X 0,Y 373.15,Z 1184.609,A -85,B 0,C 180,E1 18536.515,E2 18536.515} C_VEL
LIN {X 0,Y 373.287,Z 1188.039,A -85,B 0,C 180,E1 18542.318,E2 18542.318} C_VEL
LIN {X 0,Y 374.038,Z 1186.961,A -85,B 0,C 180,E1 18546.959,E2 18546.959} C_VEL
LIN {X 0,Y 376.125,Z 1181.093,A -85,B 0,C 180,E1 18552.763,E2 18552.763} C_VEL
LIN {X 0,Y 380.392,Z 1169.97,A -85,B 0,C 180,E1 18558.527,E2 18558.527} C_VEL
LIN {X 0,Y 387.355,Z 1153.172,A -85,B 0,C 180,E1 18564.178,E2 18564.178} C_VEL
LIN {X 0,Y 397.624,Z 1129.977,A -85,B 0,C 180,E1 18569.604,E2 18569.604} C_VEL
LIN {X 0,Y 410.643,Z 1100.911,A -85,B 0,C 180,E1 18574.453,E2 18574.453} C_VEL
LIN {X 0,Y 426.991,Z 1064.105,A -85,B 0,C 180,E1 18578.85,E2 18578.85} C_VEL
LIN {X 0,Y 439.363,Z 1035.251,A -85,B 0,C 180,E1 18581.469,E2 18581.469} C_VEL
LIN {X 0,Y 441,Z 1029.605,A -85,B 0,C 180,E1 18582.583,E2 18582.583} C_VEL
LIN {X 0,Y 441.646,Z 1027.036,A -85,B 0,C 180,E1 18584.098,E2 18584.098} C_VEL
LIN {X 0,Y 442.118,Z 1028.78,A -85,B 0,C 180,E1 18586.129,E2 18586.129} C_VEL
LIN {X 0,Y 441.255,Z 1032.859,A -85,B 0,C 180,E1 18586.92,E2 18586.92} C_VEL
LIN {X 0,Y 424.046,Z 1074.464,A -85,B 0,C 180,E1 18589.963,E2 18589.963} C_VEL
LIN {X 0,Y 408.885,Z 1111.433,A -85,B 0,C 180,E1 18593.777,E2 18593.777} C_VEL
LIN {X 0,Y 395.903,Z 1144.218,A -85,B 0,C 180,E1 18598.37,E2 18598.37} C_VEL
LIN {X 0,Y 385.897,Z 1171.554,A -85,B 0,C 180,E1 18603.574,E2 18603.574} C_VEL
LIN {X 0,Y 379.074,Z 1192.437,A -85,B 0,C 180,E1 18608.999,E2 18608.999} C_VEL
LIN {X 0,Y 375.108,Z 1207.772,A -85,B 0,C 180,E1 18614.619,E2 18614.619} C_VEL
LIN {X 0,Y 373.386,Z 1218.289,A -85,B 0,C 180,E1 18620.706,E2 18620.706} C_VEL
LIN {X 0,Y 373.074,Z 1222.365,A -85,B 0,C 180,E1 18625.374,E2 18625.374} C_VEL
LIN {X 0,Y 373.263,Z 1222.765,A -85,B 0,C 180,E1 18630.02,E2 18630.02} C_VEL
LIN {X 0,Y 373.309,Z 1219.486,A -85,B 0,C 180,E1 18634.664,E2 18634.664} C_VEL
LIN {X 0,Y 373.602,Z 1211.139,A -85,B 0,C 180,E1 18639.918,E2 18639.918} C_VEL
LIN {X 0,Y 374.77,Z 1197.392,A -85,B 0,C 180,E1 18645.231,E2 18645.231} C_VEL
LIN {X 0,Y 377.557,Z 1177.76,A -85,B 0,C 180,E1 18650.48,E2 18650.48} C_VEL
LIN {X 0,Y 382.124,Z 1152.869,A -85,B 0,C 180,E1 18655.323,E2 18655.323} C_VEL
LIN {X 0,Y 388.171,Z 1121.899,A -85,B 0,C 180,E1 18659.778,E2 18659.778} C_VEL
LIN {X 0,Y 395.106,Z 1085.95,A -85,B 0,C 180,E1 18663.535,E2 18663.535} C_VEL
LIN {X 0,Y 401.74,Z 1047.202,A -85,B 0,C 180,E1 18666.433,E2 18666.433} C_VEL
LIN {X 0,Y 405.245,Z 1023.527,A -85,B 0,C 180,E1 18667.743,E2 18667.743} C_VEL
LIN {X 0,Y 403.425,Z 1017.493,A -85,B 0,C 180,E1 18668.211,E2 18668.211} C_VEL
LIN {X 0,Y 394.267,Z 1006.08,A -85,B 0,C 180,E1 18669.42,E2 18669.42} C_VEL
LIN {X 0,Y 377.922,Z 961.291,A -85,B 0,C 180,E1 18672.466,E2 18672.466} C_VEL
LIN {X 0,Y 362.618,Z 923.03,A -85,B 0,C 180,E1 18675.131,E2 18675.131} C_VEL
LIN {X 0,Y 362.637,Z 923.03,A -85,B 0,C 180,E1 18682.374,E2 18682.374} C_VEL
LIN {X 0,Y 362.919,Z 923.03,A -85,B 0,C 180,E1 18690.026,E2 18690.026} C_VEL
LIN {X 0,Y 363.109,Z 923.801,A -85,B 0,C 180,E1 18694.21,E2 18694.21} C_VEL
LIN {X 0,Y 365.983,Z 929.122,A -85,B 0,C 180,E1 18695.401,E2 18695.401} C_VEL
LIN {X 0,Y 368.311,Z 932.775,A -85,B 0,C 180,E1 18696.241,E2 18696.241} C_VEL
LIN {X 0,Y 377.863,Z 948.154,A -85,B 0,C 180,E1 18699.185,E2 18699.185} C_VEL
LIN {X 0,Y 388.813,Z 971.031,A -85,B 0,C 180,E1 18702.092,E2 18702.092} C_VEL
LIN {X 0,Y 394.262,Z 989.025,A -85,B 0,C 180,E1 18703.578,E2 18703.578} C_VEL
LIN {X 0,Y 392.092,Z 1024.028,A -85,B 0,C 180,E1 18704.924,E2 18704.924} C_VEL
LIN {X 0,Y 388.889,Z 1051.668,A -85,B 0,C 180,E1 18706.806,E2 18706.806} C_VEL
LIN {X 0,Y 384.466,Z 1076.398,A -85,B 0,C 180,E1 18709.429,E2 18709.429} C_VEL
LIN {X 0,Y 379.871,Z 1096.187,A -85,B 0,C 180,E1 18712.574,E2 18712.574} C_VEL
LIN {X 0,Y 375.692,Z 1110.483,A -85,B 0,C 180,E1 18715.966,E2 18715.966} C_VEL
LIN {X 0,Y 371.86,Z 1120.851,A -85,B 0,C 180,E1 18720.002,E2 18720.002} C_VEL
LIN {X 0,Y 370.291,Z 1124.189,A -85,B 0,C 180,E1 18722.341,E2 18722.341} C_VEL
LIN {X 0,Y 369.019,Z 1125.889,A -85,B 0,C 180,E1 18724.7,E2 18724.7} C_VEL
LIN {X 0,Y 368.074,Z 1125.876,A -85,B 0,C 180,E1 18727.077,E2 18727.077} C_VEL
LIN {X 0,Y 367.441,Z 1121.739,A -85,B 0,C 180,E1 18731.267,E2 18731.267} C_VEL
LIN {X 0,Y 367.654,Z 1111.68,A -85,B 0,C 180,E1 18735.636,E2 18735.636} C_VEL
LIN {X 0,Y 368.559,Z 1096.369,A -85,B 0,C 180,E1 18739.594,E2 18739.594} C_VEL
LIN {X 0,Y 370.119,Z 1074.763,A -85,B 0,C 180,E1 18743.289,E2 18743.289} C_VEL
LIN {X 0,Y 371.875,Z 1049.085,A -85,B 0,C 180,E1 18746.228,E2 18746.228} C_VEL
LIN {X 0,Y 373.484,Z 1019.914,A -85,B 0,C 180,E1 18748.394,E2 18748.394} C_VEL
LIN {X 0,Y 374.367,Z 988.394,A -85,B 0,C 180,E1 18749.709,E2 18749.709} C_VEL
LIN {X 0,Y 373.476,Z 971.424,A -85,B 0,C 180,E1 18750.181,E2 18750.181} C_VEL
LIN {X 0,Y 363.103,Z 923.03,A -85,B 0,C 180,E1 18751.834,E2 18751.834} C_VEL
LIN {X 0,Y 362.566,Z 923.03,A -85,B 0,C 180,E1 18758.698,E2 18758.698} C_VEL
LIN {X 0,Y 362.563,Z 923.03,A -85,B 0,C 180,E1 18765.119,E2 18765.119} C_VEL
LIN {X 0,Y 362.633,Z 923.03,A -85,B 0,C 180,E1 18772.352,E2 18772.352} C_VEL
LIN {X 0,Y 362.944,Z 923.03,A -85,B 0,C 180,E1 18780.004,E2 18780.004} C_VEL
LIN {X 0,Y 363.295,Z 923.03,A -85,B 0,C 180,E1 18787.995,E2 18787.995} C_VEL
LIN {X 0,Y 363.748,Z 923.03,A -85,B 0,C 180,E1 18795.546,E2 18795.546} C_VEL
LIN {X 0,Y 364.33,Z 923.03,A -85,B 0,C 180,E1 18802.832,E2 18802.832} C_VEL
LIN {X 0,Y 364.975,Z 923.03,A -85,B 0,C 180,E1 18809.979,E2 18809.979} C_VEL
LIN {X 0,Y 364.355,Z 923.03,A -85,B 0,C 180,E1 18817.125,E2 18817.125} C_VEL
LIN {X 0,Y 363.815,Z 923.03,A -85,B 0,C 180,E1 18824.408,E2 18824.408} C_VEL
LIN {X 0,Y 363.29,Z 923.03,A -85,B 0,C 180,E1 18831.96,E2 18831.96} C_VEL
LIN {X 0,Y 362.952,Z 923.03,A -85,B 0,C 180,E1 18839.946,E2 18839.946} C_VEL
LIN {X 0,Y 362.66,Z 923.03,A -85,B 0,C 180,E1 18847.654,E2 18847.654} C_VEL
LIN {X 0,Y 362.617,Z 923.03,A -85,B 0,C 180,E1 18855.072,E2 18855.072} C_VEL
LIN {X 0,Y 362.713,Z 923.03,A -85,B 0,C 180,E1 18856.047,E2 18856.047} C_VEL
LIN {X 0,Y 379.834,Z 969.241,A -85,B 0,C 180,E1 18859.419,E2 18859.419} C_VEL
LIN {X 0,Y 391.99,Z 1009.713,A -85,B 0,C 180,E1 18862.869,E2 18862.869} C_VEL
LIN {X 0,Y 394.162,Z 1021.381,A -85,B 0,C 180,E1 18863.917,E2 18863.917} C_VEL
LIN {X 0,Y 387.542,Z 1059.098,A -85,B 0,C 180,E1 18867.078,E2 18867.078} C_VEL
LIN {X 0,Y 380.832,Z 1093.315,A -85,B 0,C 180,E1 18871.023,E2 18871.023} C_VEL
LIN {X 0,Y 374.696,Z 1123.349,A -85,B 0,C 180,E1 18875.762,E2 18875.762} C_VEL
LIN {X 0,Y 370.142,Z 1147.388,A -85,B 0,C 180,E1 18880.935,E2 18880.935} C_VEL
LIN {X 0,Y 367.213,Z 1165.429,A -85,B 0,C 180,E1 18886.311,E2 18886.311} C_VEL
LIN {X 0,Y 365.775,Z 1178.038,A -85,B 0,C 180,E1 18891.803,E2 18891.803} C_VEL
LIN {X 0,Y 365.3,Z 1185.879,A -85,B 0,C 180,E1 18897.627,E2 18897.627} C_VEL
LIN {X 0,Y 365.397,Z 1188.437,A -85,B 0,C 180,E1 18902.368,E2 18902.368} C_VEL
LIN {X 0,Y 366.531,Z 1186.777,A -85,B 0,C 180,E1 18908.51,E2 18908.51} C_VEL
LIN {X 0,Y 369.119,Z 1180.299,A -85,B 0,C 180,E1 18914.216,E2 18914.216} C_VEL
LIN {X 0,Y 374.876,Z 1167.012,A -85,B 0,C 180,E1 18920.65,E2 18920.65} C_VEL
LIN {X 0,Y 383.804,Z 1147.792,A -85,B 0,C 180,E1 18926.603,E2 18926.603} C_VEL
LIN {X 0,Y 395.772,Z 1122.934,A -85,B 0,C 180,E1 18931.987,E2 18931.987} C_VEL
LIN {X 0,Y 410.692,Z 1092.312,A -85,B 0,C 180,E1 18936.717,E2 18936.717} C_VEL
LIN {X 0,Y 428.785,Z 1054.911,A -85,B 0,C 180,E1 18940.854,E2 18940.854} C_VEL
LIN {X 0,Y 435.921,Z 1039.678,A -85,B 0,C 180,E1 18942.213,E2 18942.213} C_VEL
LIN {X 0,Y 437.259,Z 1036.238,A -85,B 0,C 180,E1 18942.91,E2 18942.91} C_VEL
LIN {X 0,Y 437.878,Z 1034.522,A -85,B 0,C 180,E1 18943.642,E2 18943.642} C_VEL
LIN {X 0,Y 438.47,Z 1034.859,A -85,B 0,C 180,E1 18945.669,E2 18945.669} C_VEL
LIN {X 0,Y 437.56,Z 1037.704,A -85,B 0,C 180,E1 18946.147,E2 18946.147} C_VEL
LIN {X 0,Y 418.104,Z 1080.262,A -85,B 0,C 180,E1 18949.446,E2 18949.446} C_VEL
LIN {X 0,Y 402.081,Z 1116.218,A -85,B 0,C 180,E1 18953.4,E2 18953.4} C_VEL
LIN {X 0,Y 388.112,Z 1149.052,A -85,B 0,C 180,E1 18958.317,E2 18958.317} C_VEL
LIN {X 0,Y 377.501,Z 1176.055,A -85,B 0,C 180,E1 18963.901,E2 18963.901} C_VEL
LIN {X 0,Y 370.508,Z 1196.34,A -85,B 0,C 180,E1 18969.718,E2 18969.718} C_VEL
LIN {X 0,Y 366.755,Z 1210.706,A -85,B 0,C 180,E1 18975.71,E2 18975.71} C_VEL
LIN {X 0,Y 365.353,Z 1219.387,A -85,B 0,C 180,E1 18981.699,E2 18981.699} C_VEL
LIN {X 0,Y 365.231,Z 1222.56,A -85,B 0,C 180,E1 18987.65,E2 18987.65} C_VEL
LIN {X 0,Y 365.384,Z 1220.978,A -85,B 0,C 180,E1 18992.391,E2 18992.391} C_VEL
LIN {X 0,Y 365.528,Z 1215.586,A -85,B 0,C 180,E1 18997.199,E2 18997.199} C_VEL
LIN {X 0,Y 366.137,Z 1204.762,A -85,B 0,C 180,E1 19002.534,E2 19002.534} C_VEL
LIN {X 0,Y 368.253,Z 1187.052,A -85,B 0,C 180,E1 19008.253,E2 19008.253} C_VEL
LIN {X 0,Y 372.355,Z 1163.202,A -85,B 0,C 180,E1 19013.645,E2 19013.645} C_VEL
LIN {X 0,Y 377.962,Z 1134.891,A -85,B 0,C 180,E1 19018.326,E2 19018.326} C_VEL
LIN {X 0,Y 384.597,Z 1101.914,A -85,B 0,C 180,E1 19022.356,E2 19022.356} C_VEL
LIN {X 0,Y 391.692,Z 1063.611,A -85,B 0,C 180,E1 19025.745,E2 19025.745} C_VEL
LIN {X 0,Y 398.114,Z 1022.989,A -85,B 0,C 180,E1 19028.231,E2 19028.231} C_VEL
LIN {X 0,Y 397.282,Z 1015.488,A -85,B 0,C 180,E1 19028.719,E2 19028.719} C_VEL
LIN {X 0,Y 394.267,Z 1006.08,A -85,B 0,C 180,E1 19029.42,E2 19029.42} C_VEL
LIN {X 0,Y 388.518,Z 996.029,A -85,B 0,C 180,E1 19030.323,E2 19030.323} C_VEL
LIN {X 0,Y 378.005,Z 981.924,A -85,B 0,C 180,E1 19031.709,E2 19031.709} C_VEL
LIN {X 0,Y 377.197,Z 980.089,A -85,B 0,C 180,E1 19031.849,E2 19031.849} C_VEL
LIN {X 0,Y 354.614,Z 923.03,A -85,B 0,C 180,E1 19035.876,E2 19035.876} C_VEL
LIN {X 0,Y 354.72,Z 923.03,A -85,B 0,C 180,E1 19043.391,E2 19043.391} C_VEL
LIN {X 0,Y 355.063,Z 923.607,A -85,B 0,C 180,E1 19051.418,E2 19051.418} C_VEL
LIN {X 0,Y 357.534,Z 928.743,A -85,B 0,C 180,E1 19052.807,E2 19052.807} C_VEL
LIN {X 0,Y 360.025,Z 931.591,A -85,B 0,C 180,E1 19053.853,E2 19053.853} C_VEL
LIN {X 0,Y 367.874,Z 943.897,A -85,B 0,C 180,E1 19056.822,E2 19056.822} C_VEL
LIN {X 0,Y 378.327,Z 963.076,A -85,B 0,C 180,E1 19060.015,E2 19060.015} C_VEL
LIN {X 0,Y 387.262,Z 985.81,A -85,B 0,C 180,E1 19062.477,E2 19062.477} C_VEL
LIN {X 0,Y 388.292,Z 992.169,A -85,B 0,C 180,E1 19062.881,E2 19062.881} C_VEL
LIN {X 0,Y 386.098,Z 1024.653,A -85,B 0,C 180,E1 19064.175,E2 19064.175} C_VEL
LIN {X 0,Y 382.542,Z 1053.224,A -85,B 0,C 180,E1 19066.147,E2 19066.147} C_VEL
LIN {X 0,Y 378.023,Z 1076.906,A -85,B 0,C 180,E1 19068.692,E2 19068.692} C_VEL
LIN {X 0,Y 372.793,Z 1098.157,A -85,B 0,C 180,E1 19072.14,E2 19072.14} C_VEL
LIN {X 0,Y 368.03,Z 1113.009,A -85,B 0,C 180,E1 19075.882,E2 19075.882} C_VEL
LIN {X 0,Y 364.076,Z 1122.727,A -85,B 0,C 180,E1 19080.003,E2 19080.003} C_VEL
LIN {X 0,Y 362.471,Z 1125.758,A -85,B 0,C 180,E1 19082.392,E2 19082.392} C_VEL
LIN {X 0,Y 361.139,Z 1127.065,A -85,B 0,C 180,E1 19084.803,E2 19084.803} C_VEL
LIN {X 0,Y 359.943,Z 1126.08,A -85,B 0,C 180,E1 19088.246,E2 19088.246} C_VEL
LIN {X 0,Y 359.603,Z 1119.715,A -85,B 0,C 180,E1 19092.748,E2 19092.748} C_VEL
LIN {X 0,Y 360.07,Z 1107.535,A -85,B 0,C 180,E1 19097.086,E2 19097.086} C_VEL
LIN {X 0,Y 361.271,Z 1089.324,A -85,B 0,C 180,E1 19101.15,E2 19101.15} C_VEL
LIN {X 0,Y 362.961,Z 1066.087,A -85,B 0,C 180,E1 19104.606,E2 19104.606} C_VEL
LIN {X 0,Y 364.751,Z 1038.246,A -85,B 0,C 180,E1 19107.36,E2 19107.36} C_VEL
LIN {X 0,Y 366.088,Z 1008.706,A -85,B 0,C 180,E1 19109.185,E2 19109.185} C_VEL
LIN {X 0,Y 366.104,Z 974.325,A -85,B 0,C 180,E1 19110.322,E2 19110.322} C_VEL
LIN {X 0,Y 355.121,Z 923.03,A -85,B 0,C 180,E1 19112.195,E2 19112.195} C_VEL
LIN {X 0,Y 354.569,Z 923.03,A -85,B 0,C 180,E1 19119.877,E2 19119.877} C_VEL
LIN {X 0,Y 354.552,Z 923.03,A -85,B 0,C 180,E1 19126.982,E2 19126.982} C_VEL
LIN {X 0,Y 354.707,Z 923.03,A -85,B 0,C 180,E1 19134.044,E2 19134.044} C_VEL
LIN {X 0,Y 355.107,Z 923.03,A -85,B 0,C 180,E1 19142.068,E2 19142.068} C_VEL
LIN {X 0,Y 355.48,Z 923.03,A -85,B 0,C 180,E1 19150.098,E2 19150.098} C_VEL
LIN {X 0,Y 355.989,Z 923.03,A -85,B 0,C 180,E1 19157.726,E2 19157.726} C_VEL
LIN {X 0,Y 356.65,Z 923.03,A -85,B 0,C 180,E1 19165.118,E2 19165.118} C_VEL
LIN {X 0,Y 357.071,Z 923.03,A -85,B 0,C 180,E1 19169.979,E2 19169.979} C_VEL
LIN {X 0,Y 356.419,Z 923.03,A -85,B 0,C 180,E1 19177.285,E2 19177.285} C_VEL
LIN {X 0,Y 355.868,Z 923.03,A -85,B 0,C 180,E1 19184.737,E2 19184.737} C_VEL
LIN {X 0,Y 355.337,Z 923.03,A -85,B 0,C 180,E1 19192.478,E2 19192.478} C_VEL
LIN {X 0,Y 355.088,Z 923.03,A -85,B 0,C 180,E1 19197.885,E2 19197.885} C_VEL
LIN {X 0,Y 354.758,Z 923.03,A -85,B 0,C 180,E1 19205.967,E2 19205.967} C_VEL
LIN {X 0,Y 354.598,Z 923.03,A -85,B 0,C 180,E1 19213.574,E2 19213.574} C_VEL
LIN {X 0,Y 354.793,Z 923.792,A -85,B 0,C 180,E1 19215.374,E2 19215.374} C_VEL
LIN {X 0,Y 371.731,Z 968.77,A -85,B 0,C 180,E1 19218.762,E2 19218.762} C_VEL
LIN {X 0,Y 383.791,Z 1008.47,A -85,B 0,C 180,E1 19222.214,E2 19222.214} C_VEL
LIN {X 0,Y 386.691,Z 1023.075,A -85,B 0,C 180,E1 19223.565,E2 19223.565} C_VEL
LIN {X 0,Y 379.958,Z 1060.395,A -85,B 0,C 180,E1 19226.778,E2 19226.778} C_VEL
LIN {X 0,Y 372.911,Z 1095.136,A -85,B 0,C 180,E1 19230.902,E2 19230.902} C_VEL
LIN {X 0,Y 366.785,Z 1124.464,A -85,B 0,C 180,E1 19235.668,E2 19235.668} C_VEL
LIN {X 0,Y 362.282,Z 1147.849,A -85,B 0,C 180,E1 19240.821,E2 19240.821} C_VEL
LIN {X 0,Y 359.435,Z 1165.059,A -85,B 0,C 180,E1 19246.008,E2 19246.008} C_VEL
LIN {X 0,Y 357.924,Z 1177.76,A -85,B 0,C 180,E1 19251.5,E2 19251.5} C_VEL
LIN {X 0,Y 357.427,Z 1186.091,A -85,B 0,C 180,E1 19257.574,E2 19257.574} C_VEL
LIN {X 0,Y 357.522,Z 1188.833,A -85,B 0,C 180,E1 19262.42,E2 19262.42} C_VEL
LIN {X 0,Y 358.379,Z 1188.282,A -85,B 0,C 180,E1 19267.264,E2 19267.264} C_VEL
LIN {X 0,Y 360.75,Z 1183.02,A -85,B 0,C 180,E1 19273.317,E2 19273.317} C_VEL
LIN {X 0,Y 366.234,Z 1171.249,A -85,B 0,C 180,E1 19279.898,E2 19279.898} C_VEL
LIN {X 0,Y 374.376,Z 1154.876,A -85,B 0,C 180,E1 19285.713,E2 19285.713} C_VEL
LIN {X 0,Y 386.053,Z 1132.472,A -85,B 0,C 180,E1 19291.238,E2 19291.238} C_VEL
LIN {X 0,Y 401.524,Z 1103.32,A -85,B 0,C 180,E1 19296.349,E2 19296.349} C_VEL
LIN {X 0,Y 420.574,Z 1067.45,A -85,B 0,C 180,E1 19300.801,E2 19300.801} C_VEL
LIN {X 0,Y 433.123,Z 1043.477,A -85,B 0,C 180,E1 19303.127,E2 19303.127} C_VEL
LIN {X 0,Y 434.119,Z 1041.331,A -85,B 0,C 180,E1 19304.117,E2 19304.117} C_VEL
LIN {X 0,Y 434.493,Z 1041.562,A -85,B 0,C 180,E1 19305.274,E2 19305.274} C_VEL
LIN {X 0,Y 412.782,Z 1085.044,A -85,B 0,C 180,E1 19308.81,E2 19308.81} C_VEL
LIN {X 0,Y 395.079,Z 1121.346,A -85,B 0,C 180,E1 19313.054,E2 19313.054} C_VEL
LIN {X 0,Y 380.223,Z 1153.606,A -85,B 0,C 180,E1 19318.252,E2 19318.252} C_VEL
LIN {X 0,Y 368.979,Z 1180.514,A -85,B 0,C 180,E1 19324.281,E2 19324.281} C_VEL
LIN {X 0,Y 361.942,Z 1200.029,A -85,B 0,C 180,E1 19330.513,E2 19330.513} C_VEL
LIN {X 0,Y 358.522,Z 1212.974,A -85,B 0,C 180,E1 19336.682,E2 19336.682} C_VEL
LIN {X 0,Y 357.394,Z 1220.23,A -85,B 0,C 180,E1 19342.735,E2 19342.735} C_VEL
LIN {X 0,Y 357.364,Z 1222.087,A -85,B 0,C 180,E1 19347.598,E2 19347.598} C_VEL
LIN {X 0,Y 357.514,Z 1220.362,A -85,B 0,C 180,E1 19352.444,E2 19352.444} C_VEL
LIN {X 0,Y 357.673,Z 1213.812,A -85,B 0,C 180,E1 19357.913,E2 19357.913} C_VEL
LIN {X 0,Y 358.448,Z 1202.461,A -85,B 0,C 180,E1 19363.277,E2 19363.277} C_VEL
LIN {X 0,Y 360.622,Z 1185.604,A -85,B 0,C 180,E1 19368.654,E2 19368.654} C_VEL
LIN {X 0,Y 364.59,Z 1162.997,A -85,B 0,C 180,E1 19373.841,E2 19373.841} C_VEL
LIN {X 0,Y 370.366,Z 1134.322,A -85,B 0,C 180,E1 19378.674,E2 19378.674} C_VEL
LIN {X 0,Y 377.303,Z 1100.776,A -85,B 0,C 180,E1 19382.832,E2 19382.832} C_VEL
LIN {X 0,Y 384.509,Z 1062.685,A -85,B 0,C 180,E1 19386.236,E2 19386.236} C_VEL
LIN {X 0,Y 390.976,Z 1022.651,A -85,B 0,C 180,E1 19388.722,E2 19388.722} C_VEL
LIN {X 0,Y 379.553,Z 986.64,A -85,B 0,C 180,E1 19391.394,E2 19391.394} C_VEL
LIN {X 0,Y 377.197,Z 980.089,A -85,B 0,C 180,E1 19391.849,E2 19391.849} C_VEL
LIN {X 0,Y 368.359,Z 967.122,A -85,B 0,C 180,E1 19393.05,E2 19393.05} C_VEL
LIN {X 0,Y 359.145,Z 954.271,A -85,B 0,C 180,E1 19394.275,E2 19394.275} C_VEL
LIN {X 0,Y 346.688,Z 923.03,A -85,B 0,C 180,E1 19396.613,E2 19396.613} C_VEL
LIN {X 0,Y 346.665,Z 923.03,A -85,B 0,C 180,E1 19402.396,E2 19402.396} C_VEL
LIN {X 0,Y 346.89,Z 923.824,A -85,B 0,C 180,E1 19407.205,E2 19407.205} C_VEL
LIN {X 0,Y 350.169,Z 929.322,A -85,B 0,C 180,E1 19409.85,E2 19409.85} C_VEL
LIN {X 0,Y 352.352,Z 931.487,A -85,B 0,C 180,E1 19411.075,E2 19411.075} C_VEL
LIN {X 0,Y 357.431,Z 939.552,A -85,B 0,C 180,E1 19413.648,E2 19413.648} C_VEL
LIN {X 0,Y 364.527,Z 950.841,A -85,B 0,C 180,E1 19416.441,E2 19416.441} C_VEL
LIN {X 0,Y 373.925,Z 968.597,A -85,B 0,C 180,E1 19419.473,E2 19419.473} C_VEL
LIN {X 0,Y 382.043,Z 990.146,A -85,B 0,C 180,E1 19421.877,E2 19421.877} C_VEL
LIN {X 0,Y 382.005,Z 1001.286,A -85,B 0,C 180,E1 19422.35,E2 19422.35} C_VEL
LIN {X 0,Y 379.596,Z 1032.056,A -85,B 0,C 180,E1 19423.757,E2 19423.757} C_VEL
LIN {X 0,Y 375.481,Z 1059.307,A -85,B 0,C 180,E1 19425.881,E2 19425.881} C_VEL
LIN {X 0,Y 370.662,Z 1081.976,A -85,B 0,C 180,E1 19428.539,E2 19428.539} C_VEL
LIN {X 0,Y 365.304,Z 1101.432,A -85,B 0,C 180,E1 19431.977,E2 19431.977} C_VEL
LIN {X 0,Y 360.402,Z 1115.571,A -85,B 0,C 180,E1 19435.795,E2 19435.795} C_VEL
LIN {X 0,Y 356.283,Z 1124.573,A -85,B 0,C 180,E1 19440.003,E2 19440.003} C_VEL
LIN {X 0,Y 354.633,Z 1127.208,A -85,B 0,C 180,E1 19442.445,E2 19442.445} C_VEL
LIN {X 0,Y 353.246,Z 1128.216,A -85,B 0,C 180,E1 19444.911,E2 19444.911} C_VEL
LIN {X 0,Y 351.953,Z 1126.225,A -85,B 0,C 180,E1 19448.966,E2 19448.966} C_VEL
LIN {X 0,Y 351.73,Z 1118.264,A -85,B 0,C 180,E1 19453.67,E2 19453.67} C_VEL
LIN {X 0,Y 352.328,Z 1104.837,A -85,B 0,C 180,E1 19457.981,E2 19457.981} C_VEL
LIN {X 0,Y 353.698,Z 1085.771,A -85,B 0,C 180,E1 19461.954,E2 19461.954} C_VEL
LIN {X 0,Y 355.562,Z 1060.938,A -85,B 0,C 180,E1 19465.408,E2 19465.408} C_VEL
LIN {X 0,Y 357.366,Z 1031.907,A -85,B 0,C 180,E1 19468.05,E2 19468.05} C_VEL
LIN {X 0,Y 358.586,Z 1000.143,A -85,B 0,C 180,E1 19469.764,E2 19469.764} C_VEL
LIN {X 0,Y 358.297,Z 974.911,A -85,B 0,C 180,E1 19470.538,E2 19470.538} C_VEL
LIN {X 0,Y 347.156,Z 923.03,A -85,B 0,C 180,E1 19472.456,E2 19472.456} C_VEL
LIN {X 0,Y 346.562,Z 923.03,A -85,B 0,C 180,E1 19480.85,E2 19480.85} C_VEL
LIN {X 0,Y 346.569,Z 923.03,A -85,B 0,C 180,E1 19487.84,E2 19487.84} C_VEL
LIN {X 0,Y 346.822,Z 923.03,A -85,B 0,C 180,E1 19495.881,E2 19495.881} C_VEL
LIN {X 0,Y 347.073,Z 923.03,A -85,B 0,C 180,E1 19501.363,E2 19501.363} C_VEL
LIN {X 0,Y 347.342,Z 923.03,A -85,B 0,C 180,E1 19506.928,E2 19506.928} C_VEL
LIN {X 0,Y 347.828,Z 923.03,A -85,B 0,C 180,E1 19514.869,E2 19514.869} C_VEL
LIN {X 0,Y 348.456,Z 923.03,A -85,B 0,C 180,E1 19522.503,E2 19522.503} C_VEL
LIN {X 0,Y 349.168,Z 923.03,A -85,B 0,C 180,E1 19529.978,E2 19529.978} C_VEL
LIN {X 0,Y 348.512,Z 923.03,A -85,B 0,C 180,E1 19537.451,E2 19537.451} C_VEL
LIN {X 0,Y 347.904,Z 923.03,A -85,B 0,C 180,E1 19545.082,E2 19545.082} C_VEL
LIN {X 0,Y 347.341,Z 923.03,A -85,B 0,C 180,E1 19553.024,E2 19553.024} C_VEL
LIN {X 0,Y 347.015,Z 923.03,A -85,B 0,C 180,E1 19559.43,E2 19559.43} C_VEL
LIN {X 0,Y 346.851,Z 923.03,A -85,B 0,C 180,E1 19564.466,E2 19564.466} C_VEL
LIN {X 0,Y 346.624,Z 923.03,A -85,B 0,C 180,E1 19572.17,E2 19572.17} C_VEL
LIN {X 0,Y 346.774,Z 923.03,A -85,B 0,C 180,E1 19574.572,E2 19574.572} C_VEL
LIN {X 0,Y 364.352,Z 970.238,A -85,B 0,C 180,E1 19578.253,E2 19578.253} C_VEL
LIN {X 0,Y 376.189,Z 1009.468,A -85,B 0,C 180,E1 19581.755,E2 19581.755} C_VEL
LIN {X 0,Y 379.338,Z 1023.984,A -85,B 0,C 180,E1 19583.157,E2 19583.157} C_VEL
LIN {X 0,Y 372.287,Z 1062.084,A -85,B 0,C 180,E1 19586.518,E2 19586.518} C_VEL
LIN {X 0,Y 365.09,Z 1096.5,A -85,B 0,C 180,E1 19590.728,E2 19590.728} C_VEL
LIN {X 0,Y 359.05,Z 1124.853,A -85,B 0,C 180,E1 19595.44,E2 19595.44} C_VEL
LIN {X 0,Y 354.426,Z 1148.276,A -85,B 0,C 180,E1 19600.703,E2 19600.703} C_VEL
LIN {X 0,Y 351.405,Z 1166.347,A -85,B 0,C 180,E1 19606.317,E2 19606.317} C_VEL
LIN {X 0,Y 349.939,Z 1178.753,A -85,B 0,C 180,E1 19611.93,E2 19611.93} C_VEL
LIN {X 0,Y 349.525,Z 1186.293,A -85,B 0,C 180,E1 19617.52,E2 19617.52} C_VEL
LIN {X 0,Y 349.631,Z 1189.225,A -85,B 0,C 180,E1 19622.474,E2 19622.474} C_VEL
LIN {X 0,Y 350.657,Z 1188.735,A -85,B 0,C 180,E1 19627.831,E2 19627.831} C_VEL
LIN {X 0,Y 353.078,Z 1183.948,A -85,B 0,C 180,E1 19633.612,E2 19633.612} C_VEL
LIN {X 0,Y 358.901,Z 1172.69,A -85,B 0,C 180,E1 19640.323,E2 19640.323} C_VEL
LIN {X 0,Y 367.517,Z 1156.86,A -85,B 0,C 180,E1 19646.229,E2 19646.229} C_VEL
LIN {X 0,Y 380.456,Z 1133.994,A -85,B 0,C 180,E1 19652.086,E2 19652.086} C_VEL
LIN {X 0,Y 397.727,Z 1104.141,A -85,B 0,C 180,E1 19657.434,E2 19657.434} C_VEL
LIN {X 0,Y 418.552,Z 1068.421,A -85,B 0,C 180,E1 19661.903,E2 19661.903} C_VEL
LIN {X 0,Y 429.504,Z 1049.483,A -85,B 0,C 180,E1 19663.663,E2 19663.663} C_VEL
LIN {X 0,Y 430.371,Z 1048.293,A -85,B 0,C 180,E1 19664.603,E2 19664.603} C_VEL
LIN {X 0,Y 407.529,Z 1089.742,A -85,B 0,C 180,E1 19668.161,E2 19668.161} C_VEL
LIN {X 0,Y 389.385,Z 1123.92,A -85,B 0,C 180,E1 19672.351,E2 19672.351} C_VEL
LIN {X 0,Y 373.71,Z 1155.329,A -85,B 0,C 180,E1 19677.632,E2 19677.632} C_VEL
LIN {X 0,Y 361.862,Z 1181.304,A -85,B 0,C 180,E1 19683.737,E2 19683.737} C_VEL
LIN {X 0,Y 354.411,Z 1200.314,A -85,B 0,C 180,E1 19690.081,E2 19690.081} C_VEL
LIN {X 0,Y 350.685,Z 1213.102,A -85,B 0,C 180,E1 19696.504,E2 19696.504} C_VEL
LIN {X 0,Y 349.515,Z 1219.909,A -85,B 0,C 180,E1 19702.57,E2 19702.57} C_VEL
LIN {X 0,Y 349.467,Z 1221.608,A -85,B 0,C 180,E1 19707.544,E2 19707.544} C_VEL
LIN {X 0,Y 349.63,Z 1219.735,A -85,B 0,C 180,E1 19712.499,E2 19712.499} C_VEL
LIN {X 0,Y 349.804,Z 1212.931,A -85,B 0,C 180,E1 19718.092,E2 19718.092} C_VEL
LIN {X 0,Y 350.727,Z 1200.318,A -85,B 0,C 180,E1 19723.952,E2 19723.952} C_VEL
LIN {X 0,Y 353.307,Z 1181.904,A -85,B 0,C 180,E1 19729.662,E2 19729.662} C_VEL
LIN {X 0,Y 357.751,Z 1157.86,A -85,B 0,C 180,E1 19735.006,E2 19735.006} C_VEL
LIN {X 0,Y 364.032,Z 1127.677,A -85,B 0,C 180,E1 19739.897,E2 19739.897} C_VEL
LIN {X 0,Y 371.013,Z 1094.41,A -85,B 0,C 180,E1 19743.85,E2 19743.85} C_VEL
LIN {X 0,Y 378.029,Z 1057.607,A -85,B 0,C 180,E1 19747.041,E2 19747.041} C_VEL
LIN {X 0,Y 383.562,Z 1022.491,A -85,B 0,C 180,E1 19749.226,E2 19749.226} C_VEL
LIN {X 0,Y 369.62,Z 980.991,A -85,B 0,C 180,E1 19752.405,E2 19752.405} C_VEL
LIN {X 0,Y 359.145,Z 954.271,A -85,B 0,C 180,E1 19754.275,E2 19754.275} C_VEL
LIN {X 0,Y 352.125,Z 946.596,A -85,B 0,C 180,E1 19755.177,E2 19755.177} C_VEL
LIN {X 0,Y 344.94,Z 939.061,A -85,B 0,C 180,E1 19756.121,E2 19756.121} C_VEL
LIN {X 0,Y 342.559,Z 932.413,A -85,B 0,C 180,E1 19756.769,E2 19756.769} C_VEL
LIN {X 0,Y 342.691,Z 929.846,A -85,B 0,C 180,E1 19757.27,E2 19757.27} C_VEL
LIN {X 0,Y 342.26,Z 929.596,A -85,B 0,C 180,E1 19763.983,E2 19763.983} C_VEL
LIN {X 0,Y 344.706,Z 931.532,A -85,B 0,C 180,E1 19766.903,E2 19766.903} C_VEL
LIN {X 0,Y 348.763,Z 937.31,A -85,B 0,C 180,E1 19770.094,E2 19770.094} C_VEL
LIN {X 0,Y 354.729,Z 946.928,A -85,B 0,C 180,E1 19773.36,E2 19773.36} C_VEL
LIN {X 0,Y 363.287,Z 960.963,A -85,B 0,C 180,E1 19776.771,E2 19776.771} C_VEL
LIN {X 0,Y 372.677,Z 981.758,A -85,B 0,C 180,E1 19779.904,E2 19779.904} C_VEL
LIN {X 0,Y 376.909,Z 995.468,A -85,B 0,C 180,E1 19781.295,E2 19781.295} C_VEL
LIN {X 0,Y 374.303,Z 1027.805,A -85,B 0,C 180,E1 19782.659,E2 19782.659} C_VEL
LIN {X 0,Y 370.137,Z 1056.822,A -85,B 0,C 180,E1 19784.766,E2 19784.766} C_VEL
LIN {X 0,Y 364.675,Z 1081.434,A -85,B 0,C 180,E1 19787.593,E2 19787.593} C_VEL
LIN {X 0,Y 359.197,Z 1100.819,A -85,B 0,C 180,E1 19790.926,E2 19790.926} C_VEL
LIN {X 0,Y 353.438,Z 1116.365,A -85,B 0,C 180,E1 19795.097,E2 19795.097} C_VEL
LIN {X 0,Y 349.557,Z 1124.541,A -85,B 0,C 180,E1 19798.764,E2 19798.764} C_VEL
LIN {X 0,Y 346.789,Z 1128.647,A -85,B 0,C 180,E1 19802.5,E2 19802.5} C_VEL
LIN {X 0,Y 345.368,Z 1129.297,A -85,B 0,C 180,E1 19805.023,E2 19805.023} C_VEL
LIN {X 0,Y 344.07,Z 1126.758,A -85,B 0,C 180,E1 19809.173,E2 19809.173} C_VEL
LIN {X 0,Y 343.856,Z 1118.648,A -85,B 0,C 180,E1 19813.746,E2 19813.746} C_VEL
LIN {X 0,Y 344.422,Z 1105.836,A -85,B 0,C 180,E1 19817.888,E2 19817.888} C_VEL
LIN {X 0,Y 345.73,Z 1087.53,A -85,B 0,C 180,E1 19821.812,E2 19821.812} C_VEL
LIN {X 0,Y 347.587,Z 1063.171,A -85,B 0,C 180,E1 19825.335,E2 19825.335} C_VEL
LIN {X 0,Y 349.336,Z 1035.607,A -85,B 0,C 180,E1 19827.992,E2 19827.992} C_VEL
LIN {X 0,Y 350.716,Z 1005.777,A -85,B 0,C 180,E1 19829.767,E2 19829.767} C_VEL
LIN {X 0,Y 350.508,Z 975.871,A -85,B 0,C 180,E1 19830.751,E2 19830.751} C_VEL
LIN {X 0,Y 339.207,Z 923.03,A -85,B 0,C 180,E1 19832.757,E2 19832.757} C_VEL
LIN {X 0,Y 338.638,Z 923.03,A -85,B 0,C 180,E1 19840.632,E2 19840.632} C_VEL
LIN {X 0,Y 338.664,Z 923.03,A -85,B 0,C 180,E1 19847.962,E2 19847.962} C_VEL
LIN {X 0,Y 338.732,Z 923.03,A -85,B 0,C 180,E1 19854.53,E2 19854.53} C_VEL
LIN {X 0,Y 339.109,Z 923.03,A -85,B 0,C 180,E1 19860.626,E2 19860.626} C_VEL
LIN {X 0,Y 339.547,Z 923.03,A -85,B 0,C 180,E1 19869.122,E2 19869.122} C_VEL
LIN {X 0,Y 340.126,Z 923.03,A -85,B 0,C 180,E1 19877.144,E2 19877.144} C_VEL
LIN {X 0,Y 340.8,Z 923.03,A -85,B 0,C 180,E1 19884.89,E2 19884.89} C_VEL
LIN {X 0,Y 341.279,Z 923.03,A -85,B 0,C 180,E1 19889.978,E2 19889.978} C_VEL
LIN {X 0,Y 340.57,Z 923.03,A -85,B 0,C 180,E1 19897.626,E2 19897.626} C_VEL
LIN {X 0,Y 339.978,Z 923.03,A -85,B 0,C 180,E1 19905.442,E2 19905.442} C_VEL
LIN {X 0,Y 339.378,Z 923.03,A -85,B 0,C 180,E1 19913.597,E2 19913.597} C_VEL
LIN {X 0,Y 339.118,Z 923.03,A -85,B 0,C 180,E1 19919.322,E2 19919.322} C_VEL
LIN {X 0,Y 338.73,Z 923.03,A -85,B 0,C 180,E1 19926.579,E2 19926.579} C_VEL
LIN {X 0,Y 338.807,Z 923.03,A -85,B 0,C 180,E1 19933.825,E2 19933.825} C_VEL
LIN {X 0,Y 356.391,Z 970.001,A -85,B 0,C 180,E1 19937.581,E2 19937.581} C_VEL
LIN {X 0,Y 368.261,Z 1009.437,A -85,B 0,C 180,E1 19941.187,E2 19941.187} C_VEL
LIN {X 0,Y 371.774,Z 1026.162,A -85,B 0,C 180,E1 19942.832,E2 19942.832} C_VEL
LIN {X 0,Y 364.58,Z 1063.902,A -85,B 0,C 180,E1 19946.268,E2 19946.268} C_VEL
LIN {X 0,Y 357.269,Z 1097.809,A -85,B 0,C 180,E1 19950.545,E2 19950.545} C_VEL
LIN {X 0,Y 350.976,Z 1126.762,A -85,B 0,C 180,E1 19955.516,E2 19955.516} C_VEL
LIN {X 0,Y 346.164,Z 1151.02,A -85,B 0,C 180,E1 19961.217,E2 19961.217} C_VEL
LIN {X 0,Y 343.172,Z 1169.268,A -85,B 0,C 180,E1 19967.278,E2 19967.278} C_VEL
LIN {X 0,Y 341.828,Z 1181.739,A -85,B 0,C 180,E1 19973.629,E2 19973.629} C_VEL
LIN {X 0,Y 341.628,Z 1186.482,A -85,B 0,C 180,E1 19977.462,E2 19977.462} C_VEL
LIN {X 0,Y 341.74,Z 1189.615,A -85,B 0,C 180,E1 19982.532,E2 19982.532} C_VEL
LIN {X 0,Y 342.735,Z 1189.515,A -85,B 0,C 180,E1 19987.598,E2 19987.598} C_VEL
LIN {X 0,Y 345.416,Z 1184.894,A -85,B 0,C 180,E1 19993.92,E2 19993.92} C_VEL
LIN {X 0,Y 351.616,Z 1174.128,A -85,B 0,C 180,E1 20000.763,E2 20000.763} C_VEL
LIN {X 0,Y 361.811,Z 1157.029,A -85,B 0,C 180,E1 20007.346,E2 20007.346} C_VEL
LIN {X 0,Y 376.494,Z 1133.257,A -85,B 0,C 180,E1 20013.492,E2 20013.492} C_VEL
LIN {X 0,Y 395.205,Z 1103.695,A -85,B 0,C 180,E1 20018.761,E2 20018.761} C_VEL
LIN {X 0,Y 417.435,Z 1068.988,A -85,B 0,C 180,E1 20023.096,E2 20023.096} C_VEL
LIN {X 0,Y 423.385,Z 1059.649,A -85,B 0,C 180,E1 20023.994,E2 20023.994} C_VEL
LIN {X 0,Y 423.616,Z 1059.371,A -85,B 0,C 180,E1 20024.272,E2 20024.272} C_VEL
LIN {X 0,Y 401.238,Z 1096.499,A -85,B 0,C 180,E1 20027.717,E2 20027.717} C_VEL
LIN {X 0,Y 381.33,Z 1130.926,A -85,B 0,C 180,E1 20032.278,E2 20032.278} C_VEL
LIN {X 0,Y 364.258,Z 1162.757,A -85,B 0,C 180,E1 20038.202,E2 20038.202} C_VEL
LIN {X 0,Y 352.456,Z 1187.066,A -85,B 0,C 180,E1 20044.639,E2 20044.639} C_VEL
LIN {X 0,Y 345.833,Z 1203.561,A -85,B 0,C 180,E1 20050.895,E2 20050.895} C_VEL
LIN {X 0,Y 342.515,Z 1214.634,A -85,B 0,C 180,E1 20057.28,E2 20057.28} C_VEL
LIN {X 0,Y 341.621,Z 1219.591,A -85,B 0,C 180,E1 20062.398,E2 20062.398} C_VEL
LIN {X 0,Y 341.572,Z 1221.128,A -85,B 0,C 180,E1 20067.487,E2 20067.487} C_VEL
LIN {X 0,Y 341.749,Z 1219.081,A -85,B 0,C 180,E1 20072.556,E2 20072.556} C_VEL
LIN {X 0,Y 341.932,Z 1212.033,A -85,B 0,C 180,E1 20078.28,E2 20078.28} C_VEL
LIN {X 0,Y 342.901,Z 1199.307,A -85,B 0,C 180,E1 20084.199,E2 20084.199} C_VEL
LIN {X 0,Y 345.632,Z 1180.333,A -85,B 0,C 180,E1 20090.118,E2 20090.118} C_VEL
LIN {X 0,Y 350.363,Z 1155.812,A -85,B 0,C 180,E1 20095.571,E2 20095.571} C_VEL
LIN {X 0,Y 356.519,Z 1126.981,A -85,B 0,C 180,E1 20100.282,E2 20100.282} C_VEL
LIN {X 0,Y 363.966,Z 1092.398,A -85,B 0,C 180,E1 20104.433,E2 20104.433} C_VEL
LIN {X 0,Y 371.469,Z 1053.48,A -85,B 0,C 180,E1 20107.797,E2 20107.797} C_VEL
LIN {X 0,Y 376.304,Z 1024.941,A -85,B 0,C 180,E1 20109.57,E2 20109.57} C_VEL
LIN {X 0,Y 362.709,Z 983.953,A -85,B 0,C 180,E1 20112.825,E2 20112.825} C_VEL
LIN {X 0,Y 344.94,Z 939.061,A -85,B 0,C 180,E1 20116.121,E2 20116.121} C_VEL
LIN {X 0,Y 342.32,Z 935.82,A -85,B 0,C 180,E1 20117.032,E2 20117.032} C_VEL
LIN {X 0,Y 339.769,Z 936.833,A -85,B 0,C 180,E1 20119.973,E2 20119.973} C_VEL
LIN {X 0,Y 342.46,Z 938.454,A -85,B 0,C 180,E1 20126.399,E2 20126.399} C_VEL
LIN {X 0,Y 346.247,Z 944.599,A -85,B 0,C 180,E1 20129.713,E2 20129.713} C_VEL
LIN {X 0,Y 352.88,Z 955.508,A -85,B 0,C 180,E1 20133.447,E2 20133.447} C_VEL
LIN {X 0,Y 361.429,Z 970.912,A -85,B 0,C 180,E1 20136.938,E2 20136.938} C_VEL
LIN {X 0,Y 369.475,Z 990.676,A -85,B 0,C 180,E1 20139.753,E2 20139.753} C_VEL
LIN {X 0,Y 371.366,Z 999.088,A -85,B 0,C 180,E1 20140.517,E2 20140.517} C_VEL
LIN {X 0,Y 368.593,Z 1029.776,A -85,B 0,C 180,E1 20141.867,E2 20141.867} C_VEL
LIN {X 0,Y 364.336,Z 1057.26,A -85,B 0,C 180,E1 20143.9,E2 20143.9} C_VEL
LIN {X 0,Y 358.562,Z 1082.14,A -85,B 0,C 180,E1 20146.755,E2 20146.755} C_VEL
LIN {X 0,Y 352.718,Z 1101.538,A -85,B 0,C 180,E1 20150.135,E2 20150.135} C_VEL
LIN {X 0,Y 347.357,Z 1115.466,A -85,B 0,C 180,E1 20153.759,E2 20153.759} C_VEL
LIN {X 0,Y 342.389,Z 1125.489,A -85,B 0,C 180,E1 20158.106,E2 20158.106} C_VEL
LIN {X 0,Y 338.915,Z 1130.001,A -85,B 0,C 180,E1 20162.558,E2 20162.558} C_VEL
LIN {X 0,Y 337.463,Z 1130.291,A -85,B 0,C 180,E1 20165.141,E2 20165.141} C_VEL
LIN {X 0,Y 336.193,Z 1127.22,A -85,B 0,C 180,E1 20169.33,E2 20169.33} C_VEL
LIN {X 0,Y 335.984,Z 1118.638,A -85,B 0,C 180,E1 20173.967,E2 20173.967} C_VEL
LIN {X 0,Y 336.622,Z 1104.86,A -85,B 0,C 180,E1 20178.317,E2 20178.317} C_VEL
LIN {X 0,Y 338.039,Z 1085.43,A -85,B 0,C 180,E1 20182.335,E2 20182.335} C_VEL
LIN {X 0,Y 339.896,Z 1061.712,A -85,B 0,C 180,E1 20185.691,E2 20185.691} C_VEL
LIN {X 0,Y 341.721,Z 1032.913,A -85,B 0,C 180,E1 20188.401,E2 20188.401} C_VEL
LIN {X 0,Y 343.047,Z 1001.14,A -85,B 0,C 180,E1 20190.175,E2 20190.175} C_VEL
LIN {X 0,Y 342.556,Z 976.223,A -85,B 0,C 180,E1 20190.984,E2 20190.984} C_VEL
LIN {X 0,Y 331.271,Z 923.03,A -85,B 0,C 180,E1 20193.036,E2 20193.036} C_VEL
LIN {X 0,Y 330.709,Z 923.03,A -85,B 0,C 180,E1 20199.773,E2 20199.773} C_VEL
LIN {X 0,Y 330.71,Z 923.03,A -85,B 0,C 180,E1 20206.981,E2 20206.981} C_VEL
LIN {X 0,Y 330.777,Z 923.03,A -85,B 0,C 180,E1 20213.542,E2 20213.542} C_VEL
LIN {X 0,Y 331.119,Z 923.03,A -85,B 0,C 180,E1 20220.127,E2 20220.127} C_VEL
LIN {X 0,Y 331.552,Z 923.03,A -85,B 0,C 180,E1 20228.594,E2 20228.594} C_VEL
LIN {X 0,Y 332.16,Z 923.03,A -85,B 0,C 180,E1 20236.83,E2 20236.83} C_VEL
LIN {X 0,Y 332.886,Z 923.03,A -85,B 0,C 180,E1 20244.769,E2 20244.769} C_VEL
LIN {X 0,Y 333.375,Z 923.03,A -85,B 0,C 180,E1 20249.977,E2 20249.977} C_VEL
LIN {X 0,Y 332.63,Z 923.03,A -85,B 0,C 180,E1 20257.809,E2 20257.809} C_VEL
LIN {X 0,Y 331.997,Z 923.03,A -85,B 0,C 180,E1 20265.823,E2 20265.823} C_VEL
LIN {X 0,Y 331.602,Z 923.03,A -85,B 0,C 180,E1 20271.353,E2 20271.353} C_VEL
LIN {X 0,Y 331.135,Z 923.03,A -85,B 0,C 180,E1 20279.878,E2 20279.878} C_VEL
LIN {X 0,Y 330.852,Z 923.03,A -85,B 0,C 180,E1 20286.391,E2 20286.391} C_VEL
LIN {X 0,Y 330.814,Z 923.03,A -85,B 0,C 180,E1 20293.038,E2 20293.038} C_VEL
LIN {X 0,Y 348.415,Z 969.756,A -85,B 0,C 180,E1 20296.894,E2 20296.894} C_VEL
LIN {X 0,Y 360.296,Z 1009.157,A -85,B 0,C 180,E1 20300.577,E2 20300.577} C_VEL
LIN {X 0,Y 364.346,Z 1027.357,A -85,B 0,C 180,E1 20302.429,E2 20302.429} C_VEL
LIN {X 0,Y 356.935,Z 1065.292,A -85,B 0,C 180,E1 20305.98,E2 20305.98} C_VEL
LIN {X 0,Y 349.366,Z 1099.401,A -85,B 0,C 180,E1 20310.406,E2 20310.406} C_VEL
LIN {X 0,Y 343.228,Z 1127.051,A -85,B 0,C 180,E1 20315.273,E2 20315.273} C_VEL
LIN {X 0,Y 338.52,Z 1150.176,A -85,B 0,C 180,E1 20320.776,E2 20320.776} C_VEL
LIN {X 0,Y 335.377,Z 1168.84,A -85,B 0,C 180,E1 20326.978,E2 20326.978} C_VEL
LIN {X 0,Y 334.029,Z 1180.802,A -85,B 0,C 180,E1 20332.916,E2 20332.916} C_VEL
LIN {X 0,Y 333.64,Z 1187.725,A -85,B 0,C 180,E1 20338.7,E2 20338.7} C_VEL
LIN {X 0,Y 334.169,Z 1190.465,A -85,B 0,C 180,E1 20345.186,E2 20345.186} C_VEL
LIN {X 0,Y 335.797,Z 1189.017,A -85,B 0,C 180,E1 20350.367,E2 20350.367} C_VEL
LIN {X 0,Y 340.063,Z 1182.288,A -85,B 0,C 180,E1 20357.204,E2 20357.204} C_VEL
LIN {X 0,Y 348.463,Z 1169.097,A -85,B 0,C 180,E1 20364.243,E2 20364.243} C_VEL
LIN {X 0,Y 361.337,Z 1149.781,A -85,B 0,C 180,E1 20370.756,E2 20370.756} C_VEL
LIN {X 0,Y 379.139,Z 1123.809,A -85,B 0,C 180,E1 20376.712,E2 20376.712} C_VEL
LIN {X 0,Y 400.849,Z 1092.578,A -85,B 0,C 180,E1 20381.634,E2 20381.634} C_VEL
LIN {X 0,Y 415.068,Z 1072.355,A -85,B 0,C 180,E1 20384.124,E2 20384.124} C_VEL
LIN {X 0,Y 391.414,Z 1108.427,A -85,B 0,C 180,E1 20387.904,E2 20387.904} C_VEL
LIN {X 0,Y 369.266,Z 1144.354,A -85,B 0,C 180,E1 20393.407,E2 20393.407} C_VEL
LIN {X 0,Y 353.431,Z 1172.29,A -85,B 0,C 180,E1 20399.516,E2 20399.516} C_VEL
LIN {X 0,Y 342.793,Z 1193.206,A -85,B 0,C 180,E1 20405.963,E2 20405.963} C_VEL
LIN {X 0,Y 336.444,Z 1208.715,A -85,B 0,C 180,E1 20413.051,E2 20413.051} C_VEL
LIN {X 0,Y 334.04,Z 1217.317,A -85,B 0,C 180,E1 20419.599,E2 20419.599} C_VEL
LIN {X 0,Y 333.601,Z 1220.501,A -85,B 0,C 180,E1 20425.187,E2 20425.187} C_VEL
LIN {X 0,Y 333.879,Z 1220.005,A -85,B 0,C 180,E1 20430.023,E2 20430.023} C_VEL
LIN {X 0,Y 333.998,Z 1214.284,A -85,B 0,C 180,E1 20436.386,E2 20436.386} C_VEL
LIN {X 0,Y 334.579,Z 1203.299,A -85,B 0,C 180,E1 20442.41,E2 20442.41} C_VEL
LIN {X 0,Y 336.894,Z 1185.328,A -85,B 0,C 180,E1 20448.75,E2 20448.75} C_VEL
LIN {X 0,Y 341.191,Z 1162.488,A -85,B 0,C 180,E1 20454.389,E2 20454.389} C_VEL
LIN {X 0,Y 347.319,Z 1133.971,A -85,B 0,C 180,E1 20459.529,E2 20459.529} C_VEL
LIN {X 0,Y 354.627,Z 1100.867,A -85,B 0,C 180,E1 20463.907,E2 20463.907} C_VEL
LIN {X 0,Y 362.43,Z 1062.752,A -85,B 0,C 180,E1 20467.542,E2 20467.542} C_VEL
LIN {X 0,Y 368.566,Z 1025.479,A -85,B 0,C 180,E1 20470.07,E2 20470.07} C_VEL
LIN {X 0,Y 355.063,Z 984.719,A -85,B 0,C 180,E1 20473.417,E2 20473.417} C_VEL
LIN {X 0,Y 339.896,Z 945.338,A -85,B 0,C 180,E1 20476.475,E2 20476.475} C_VEL
LIN {X 0,Y 340.565,Z 937.382,A -85,B 0,C 180,E1 20477.877,E2 20477.877} C_VEL
LIN {X 0,Y 339.769,Z 936.833,A -85,B 0,C 180,E1 20479.973,E2 20479.973} C_VEL
LIN {X 0,Y 339.245,Z 939.293,A -85,B 0,C 180,E1 20482.149,E2 20482.149} C_VEL
LIN {X 0,Y 339.72,Z 945.392,A -85,B 0,C 180,E1 20485.349,E2 20485.349} C_VEL
LIN {X 0,Y 340.03,Z 945.62,A -85,B 0,C 180,E1 20485.715,E2 20485.715} C_VEL
LIN {X 0,Y 344.944,Z 954.01,A -85,B 0,C 180,E1 20490.174,E2 20490.174} C_VEL
LIN {X 0,Y 351.458,Z 964.902,A -85,B 0,C 180,E1 20493.738,E2 20493.738} C_VEL
LIN {X 0,Y 359.273,Z 980.573,A -85,B 0,C 180,E1 20497.02,E2 20497.02} C_VEL
LIN {X 0,Y 366.162,Z 1000.113,A -85,B 0,C 180,E1 20499.604,E2 20499.604} C_VEL
LIN {X 0,Y 362.962,Z 1032.517,A -85,B 0,C 180,E1 20501.08,E2 20501.08} C_VEL
LIN {X 0,Y 358.404,Z 1059.467,A -85,B 0,C 180,E1 20503.153,E2 20503.153} C_VEL
LIN {X 0,Y 352.276,Z 1083.856,A -85,B 0,C 180,E1 20506.04,E2 20506.04} C_VEL
LIN {X 0,Y 345.735,Z 1104.042,A -85,B 0,C 180,E1 20509.679,E2 20509.679} C_VEL
LIN {X 0,Y 339.747,Z 1118.157,A -85,B 0,C 180,E1 20513.619,E2 20513.619} C_VEL
LIN {X 0,Y 335.256,Z 1126.486,A -85,B 0,C 180,E1 20517.419,E2 20517.419} C_VEL
LIN {X 0,Y 332.553,Z 1130.121,A -85,B 0,C 180,E1 20520.427,E2 20520.427} C_VEL
LIN {X 0,Y 329.575,Z 1131.247,A -85,B 0,C 180,E1 20525.264,E2 20525.264} C_VEL
LIN {X 0,Y 328.257,Z 1127.401,A -85,B 0,C 180,E1 20529.704,E2 20529.704} C_VEL
LIN {X 0,Y 328.197,Z 1117.174,A -85,B 0,C 180,E1 20534.714,E2 20534.714} C_VEL
LIN {X 0,Y 328.957,Z 1102.262,A -85,B 0,C 180,E1 20539.104,E2 20539.104} C_VEL
LIN {X 0,Y 330.454,Z 1082.002,A -85,B 0,C 180,E1 20543.077,E2 20543.077} C_VEL
LIN {X 0,Y 332.317,Z 1057.882,A -85,B 0,C 180,E1 20546.321,E2 20546.321} C_VEL
LIN {X 0,Y 334.211,Z 1028.66,A -85,B 0,C 180,E1 20548.913,E2 20548.913} C_VEL
LIN {X 0,Y 335.39,Z 996.67,A -85,B 0,C 180,E1 20550.558,E2 20550.558} C_VEL
LIN {X 0,Y 334.917,Z 977.945,A -85,B 0,C 180,E1 20551.163,E2 20551.163} C_VEL
LIN {X 0,Y 323.292,Z 923.03,A -85,B 0,C 180,E1 20553.392,E2 20553.392} C_VEL
LIN {X 0,Y 322.676,Z 923.03,A -85,B 0,C 180,E1 20561.442,E2 20561.442} C_VEL
LIN {X 0,Y 322.699,Z 923.03,A -85,B 0,C 180,E1 20569.01,E2 20569.01} C_VEL
LIN {X 0,Y 322.916,Z 923.03,A -85,B 0,C 180,E1 20575.812,E2 20575.812} C_VEL
LIN {X 0,Y 323.323,Z 923.03,A -85,B 0,C 180,E1 20582.628,E2 20582.628} C_VEL
LIN {X 0,Y 323.749,Z 923.03,A -85,B 0,C 180,E1 20590.907,E2 20590.907} C_VEL
LIN {X 0,Y 324.401,Z 923.03,A -85,B 0,C 180,E1 20599.239,E2 20599.239} C_VEL
LIN {X 0,Y 325.249,Z 923.03,A -85,B 0,C 180,E1 20607.314,E2 20607.314} C_VEL
LIN {X 0,Y 325.236,Z 923.03,A -85,B 0,C 180,E1 20612.639,E2 20612.639} C_VEL
LIN {X 0,Y 324.463,Z 923.03,A -85,B 0,C 180,E1 20620.711,E2 20620.711} C_VEL
LIN {X 0,Y 323.788,Z 923.03,A -85,B 0,C 180,E1 20629.041,E2 20629.041} C_VEL
LIN {X 0,Y 323.312,Z 923.03,A -85,B 0,C 180,E1 20637.368,E2 20637.368} C_VEL
LIN {X 0,Y 322.967,Z 923.03,A -85,B 0,C 180,E1 20644.124,E2 20644.124} C_VEL
LIN {X 0,Y 322.807,Z 923.03,A -85,B 0,C 180,E1 20652.214,E2 20652.214} C_VEL
LIN {X 0,Y 340.008,Z 968.418,A -85,B 0,C 180,E1 20656.083,E2 20656.083} C_VEL
LIN {X 0,Y 351.889,Z 1007.147,A -85,B 0,C 180,E1 20659.77,E2 20659.77} C_VEL
LIN {X 0,Y 356.894,Z 1028.66,A -85,B 0,C 180,E1 20662.025,E2 20662.025} C_VEL
LIN {X 0,Y 349.1,Z 1067.236,A -85,B 0,C 180,E1 20665.753,E2 20665.753} C_VEL
LIN {X 0,Y 341.776,Z 1099.631,A -85,B 0,C 180,E1 20670.064,E2 20670.064} C_VEL
LIN {X 0,Y 335.368,Z 1127.77,A -85,B 0,C 180,E1 20675.122,E2 20675.122} C_VEL
LIN {X 0,Y 330.447,Z 1151.671,A -85,B 0,C 180,E1 20680.982,E2 20680.982} C_VEL
LIN {X 0,Y 327.362,Z 1170.013,A -85,B 0,C 180,E1 20687.332,E2 20687.332} C_VEL
LIN {X 0,Y 326.07,Z 1181.637,A -85,B 0,C 180,E1 20693.344,E2 20693.344} C_VEL
LIN {X 0,Y 325.773,Z 1188.966,A -85,B 0,C 180,E1 20699.997,E2 20699.997} C_VEL
LIN {X 0,Y 326.321,Z 1190.962,A -85,B 0,C 180,E1 20705.311,E2 20705.311} C_VEL
LIN {X 0,Y 328.023,Z 1189.76,A -85,B 0,C 180,E1 20710.616,E2 20710.616} C_VEL
LIN {X 0,Y 332.402,Z 1183.684,A -85,B 0,C 180,E1 20717.414,E2 20717.414} C_VEL
LIN {X 0,Y 340.935,Z 1171.588,A -85,B 0,C 180,E1 20724.444,E2 20724.444} C_VEL
LIN {X 0,Y 354.565,Z 1152.933,A -85,B 0,C 180,E1 20731.214,E2 20731.214} C_VEL
LIN {X 0,Y 373.494,Z 1127.557,A -85,B 0,C 180,E1 20737.361,E2 20737.361} C_VEL
LIN {X 0,Y 397.189,Z 1096.464,A -85,B 0,C 180,E1 20742.474,E2 20742.474} C_VEL
LIN {X 0,Y 405.441,Z 1085.72,A -85,B 0,C 180,E1 20743.841,E2 20743.841} C_VEL
LIN {X 0,Y 403.373,Z 1088.688,A -85,B 0,C 180,E1 20744.409,E2 20744.409} C_VEL
LIN {X 0,Y 379.521,Z 1122.508,A -85,B 0,C 180,E1 20748.584,E2 20748.584} C_VEL
LIN {X 0,Y 358.494,Z 1154.418,A -85,B 0,C 180,E1 20754.238,E2 20754.238} C_VEL
LIN {X 0,Y 343.074,Z 1180.018,A -85,B 0,C 180,E1 20760.687,E2 20760.687} C_VEL
LIN {X 0,Y 333.273,Z 1198.575,A -85,B 0,C 180,E1 20767.358,E2 20767.358} C_VEL
LIN {X 0,Y 328.036,Z 1210.943,A -85,B 0,C 180,E1 20773.981,E2 20773.981} C_VEL
LIN {X 0,Y 326.179,Z 1217.119,A -85,B 0,C 180,E1 20779.346,E2 20779.346} C_VEL
LIN {X 0,Y 325.714,Z 1219.999,A -85,B 0,C 180,E1 20784.7,E2 20784.7} C_VEL
LIN {X 0,Y 326.003,Z 1219.352,A -85,B 0,C 180,E1 20790.023,E2 20790.023} C_VEL
LIN {X 0,Y 326.099,Z 1214.872,A -85,B 0,C 180,E1 20795.341,E2 20795.341} C_VEL
LIN {X 0,Y 326.533,Z 1205.005,A -85,B 0,C 180,E1 20801.365,E2 20801.365} C_VEL
LIN {X 0,Y 328.373,Z 1189.448,A -85,B 0,C 180,E1 20807.427,E2 20807.427} C_VEL
LIN {X 0,Y 332.062,Z 1168.642,A -85,B 0,C 180,E1 20813.132,E2 20813.132} C_VEL
LIN {X 0,Y 337.655,Z 1142.337,A -85,B 0,C 180,E1 20818.415,E2 20818.415} C_VEL
LIN {X 0,Y 345.035,Z 1110.016,A -85,B 0,C 180,E1 20823.181,E2 20823.181} C_VEL
LIN {X 0,Y 353.135,Z 1072.328,A -85,B 0,C 180,E1 20827.176,E2 20827.176} C_VEL
LIN {X 0,Y 360.616,Z 1033.004,A -85,B 0,C 180,E1 20830.097,E2 20830.097} C_VEL
LIN {X 0,Y 360.754,Z 1025.872,A -85,B 0,C 180,E1 20830.598,E2 20830.598} C_VEL
LIN {X 0,Y 346.949,Z 984.142,A -85,B 0,C 180,E1 20834.121,E2 20834.121} C_VEL
LIN {X 0,Y 337.167,Z 957.935,A -85,B 0,C 180,E1 20836.269,E2 20836.269} C_VEL
LIN {X 0,Y 338.516,Z 944.845,A -85,B 0,C 180,E1 20838.429,E2 20838.429} C_VEL
LIN {X 0,Y 339.125,Z 945.234,A -85,B 0,C 180,E1 20844.605,E2 20844.605} C_VEL
LIN {X 0,Y 340.03,Z 945.62,A -85,B 0,C 180,E1 20845.715,E2 20845.715} C_VEL
LIN {X 0,Y 341.069,Z 948.182,A -85,B 0,C 180,E1 20847.087,E2 20847.087} C_VEL
LIN {X 0,Y 343.84,Z 963.709,A -85,B 0,C 180,E1 20850.748,E2 20850.748} C_VEL
LIN {X 0,Y 350.612,Z 976.018,A -85,B 0,C 180,E1 20854.352,E2 20854.352} C_VEL
LIN {X 0,Y 357.714,Z 992.54,A -85,B 0,C 180,E1 20857.386,E2 20857.386} C_VEL
LIN {X 0,Y 360.857,Z 1004.488,A -85,B 0,C 180,E1 20858.772,E2 20858.772} C_VEL
LIN {X 0,Y 357.404,Z 1036.148,A -85,B 0,C 180,E1 20860.314,E2 20860.314} C_VEL
LIN {X 0,Y 352.258,Z 1063.236,A -85,B 0,C 180,E1 20862.528,E2 20862.528} C_VEL
LIN {X 0,Y 345.792,Z 1086.784,A -85,B 0,C 180,E1 20865.45,E2 20865.45} C_VEL
LIN {X 0,Y 338.443,Z 1107.354,A -85,B 0,C 180,E1 20869.389,E2 20869.389} C_VEL
LIN {X 0,Y 332.131,Z 1120.844,A -85,B 0,C 180,E1 20873.472,E2 20873.472} C_VEL
LIN {X 0,Y 327.494,Z 1128.485,A -85,B 0,C 180,E1 20877.358,E2 20877.358} C_VEL
LIN {X 0,Y 325.044,Z 1131.375,A -85,B 0,C 180,E1 20880.003,E2 20880.003} C_VEL
LIN {X 0,Y 323.153,Z 1132.534,A -85,B 0,C 180,E1 20882.683,E2 20882.683} C_VEL
LIN {X 0,Y 321.129,Z 1131.229,A -85,B 0,C 180,E1 20886.759,E2 20886.759} C_VEL
LIN {X 0,Y 320.238,Z 1124.873,A -85,B 0,C 180,E1 20891.572,E2 20891.572} C_VEL
LIN {X 0,Y 320.498,Z 1112.548,A -85,B 0,C 180,E1 20896.436,E2 20896.436} C_VEL
LIN {X 0,Y 321.584,Z 1095.109,A -85,B 0,C 180,E1 20900.826,E2 20900.826} C_VEL
LIN {X 0,Y 323.344,Z 1072.849,A -85,B 0,C 180,E1 20904.62,E2 20904.62} C_VEL
LIN {X 0,Y 325.332,Z 1046.53,A -85,B 0,C 180,E1 20907.68,E2 20907.68} C_VEL
LIN {X 0,Y 326.939,Z 1016.552,A -85,B 0,C 180,E1 20909.895,E2 20909.895} C_VEL
LIN {X 0,Y 327.73,Z 981.607,A -85,B 0,C 180,E1 20911.271,E2 20911.271} C_VEL
LIN {X 0,Y 315.312,Z 923.03,A -85,B 0,C 180,E1 20913.694,E2 20913.694} C_VEL
LIN {X 0,Y 314.705,Z 923.03,A -85,B 0,C 180,E1 20922.243,E2 20922.243} C_VEL
LIN {X 0,Y 314.723,Z 923.03,A -85,B 0,C 180,E1 20930.199,E2 20930.199} C_VEL
LIN {X 0,Y 315.059,Z 923.03,A -85,B 0,C 180,E1 20938.132,E2 20938.132} C_VEL
LIN {X 0,Y 315.488,Z 923.03,A -85,B 0,C 180,E1 20945.519,E2 20945.519} C_VEL
LIN {X 0,Y 315.999,Z 923.03,A -85,B 0,C 180,E1 20953.303,E2 20953.303} C_VEL
LIN {X 0,Y 316.692,Z 923.03,A -85,B 0,C 180,E1 20961.747,E2 20961.747} C_VEL
LIN {X 0,Y 317.598,Z 923.03,A -85,B 0,C 180,E1 20969.976,E2 20969.976} C_VEL
LIN {X 0,Y 316.741,Z 923.03,A -85,B 0,C 180,E1 20978.203,E2 20978.203} C_VEL
LIN {X 0,Y 316.046,Z 923.03,A -85,B 0,C 180,E1 20986.644,E2 20986.644} C_VEL
LIN {X 0,Y 315.505,Z 923.03,A -85,B 0,C 180,E1 20994.488,E2 20994.488} C_VEL
LIN {X 0,Y 315.095,Z 923.03,A -85,B 0,C 180,E1 21001.807,E2 21001.807} C_VEL
LIN {X 0,Y 314.788,Z 923.03,A -85,B 0,C 180,E1 21009.816,E2 21009.816} C_VEL
LIN {X 0,Y 314.892,Z 923.138,A -85,B 0,C 180,E1 21011.388,E2 21011.388} C_VEL
LIN {X 0,Y 332.142,Z 968.582,A -85,B 0,C 180,E1 21015.383,E2 21015.383} C_VEL
LIN {X 0,Y 344.141,Z 1007.482,A -85,B 0,C 180,E1 21019.196,E2 21019.196} C_VEL
LIN {X 0,Y 349.481,Z 1029.659,A -85,B 0,C 180,E1 21021.588,E2 21021.588} C_VEL
LIN {X 0,Y 341.718,Z 1067.237,A -85,B 0,C 180,E1 21025.292,E2 21025.292} C_VEL
LIN {X 0,Y 334.089,Z 1100.2,A -85,B 0,C 180,E1 21029.766,E2 21029.766} C_VEL
LIN {X 0,Y 327.337,Z 1129.293,A -85,B 0,C 180,E1 21035.146,E2 21035.146} C_VEL
LIN {X 0,Y 322.361,Z 1153.094,A -85,B 0,C 180,E1 21041.197,E2 21041.197} C_VEL
LIN {X 0,Y 319.339,Z 1171.098,A -85,B 0,C 180,E1 21047.702,E2 21047.702} C_VEL
LIN {X 0,Y 318.212,Z 1181.468,A -85,B 0,C 180,E1 21053.179,E2 21053.179} C_VEL
LIN {X 0,Y 317.871,Z 1188.054,A -85,B 0,C 180,E1 21058.635,E2 21058.635} C_VEL
LIN {X 0,Y 318.471,Z 1191.46,A -85,B 0,C 180,E1 21065.442,E2 21065.442} C_VEL
LIN {X 0,Y 320.274,Z 1190.516,A -85,B 0,C 180,E1 21070.875,E2 21070.875} C_VEL
LIN {X 0,Y 324.929,Z 1184.871,A -85,B 0,C 180,E1 21077.828,E2 21077.828} C_VEL
LIN {X 0,Y 333.99,Z 1173.262,A -85,B 0,C 180,E1 21085.03,E2 21085.03} C_VEL
LIN {X 0,Y 348.759,Z 1154.924,A -85,B 0,C 180,E1 21092.047,E2 21092.047} C_VEL
LIN {X 0,Y 368.922,Z 1130.154,A -85,B 0,C 180,E1 21098.278,E2 21098.278} C_VEL
LIN {X 0,Y 393.553,Z 1100.713,A -85,B 0,C 180,E1 21103.299,E2 21103.299} C_VEL
LIN {X 0,Y 396.827,Z 1096.742,A -85,B 0,C 180,E1 21103.83,E2 21103.83} C_VEL
LIN {X 0,Y 367.351,Z 1135.535,A -85,B 0,C 180,E1 21109.37,E2 21109.37} C_VEL
LIN {X 0,Y 345.476,Z 1166.757,A -85,B 0,C 180,E1 21115.907,E2 21115.907} C_VEL
LIN {X 0,Y 331.177,Z 1189.636,A -85,B 0,C 180,E1 21122.881,E2 21122.881} C_VEL
LIN {X 0,Y 322.822,Z 1205.338,A -85,B 0,C 180,E1 21129.95,E2 21129.95} C_VEL
LIN {X 0,Y 318.672,Z 1215.781,A -85,B 0,C 180,E1 21137.705,E2 21137.705} C_VEL
LIN {X 0,Y 317.816,Z 1219.603,A -85,B 0,C 180,E1 21144.568,E2 21144.568} C_VEL
LIN {X 0,Y 318.152,Z 1218.67,A -85,B 0,C 180,E1 21150.024,E2 21150.024} C_VEL
LIN {X 0,Y 318.25,Z 1214,A -85,B 0,C 180,E1 21155.473,E2 21155.473} C_VEL
LIN {X 0,Y 318.708,Z 1203.824,A -85,B 0,C 180,E1 21161.648,E2 21161.648} C_VEL
LIN {X 0,Y 320.7,Z 1187.884,A -85,B 0,C 180,E1 21167.858,E2 21167.858} C_VEL
LIN {X 0,Y 324.55,Z 1166.643,A -85,B 0,C 180,E1 21173.7,E2 21173.7} C_VEL
LIN {X 0,Y 330.5,Z 1139.856,A -85,B 0,C 180,E1 21179.088,E2 21179.088} C_VEL
LIN {X 0,Y 338.318,Z 1106.408,A -85,B 0,C 180,E1 21183.988,E2 21183.988} C_VEL
LIN {X 0,Y 346.187,Z 1069.953,A -85,B 0,C 180,E1 21187.837,E2 21187.837} C_VEL
LIN {X 0,Y 353.75,Z 1030.823,A -85,B 0,C 180,E1 21190.746,E2 21190.746} C_VEL
LIN {X 0,Y 342.408,Z 993.636,A -85,B 0,C 180,E1 21194.018,E2 21194.018} C_VEL
LIN {X 0,Y 334.394,Z 971.114,A -85,B 0,C 180,E1 21195.972,E2 21195.972} C_VEL
LIN {X 0,Y 336.47,Z 952.391,A -85,B 0,C 180,E1 21199.062,E2 21199.062} C_VEL
LIN {X 0,Y 338.255,Z 953.354,A -85,B 0,C 180,E1 21205.743,E2 21205.743} C_VEL
LIN {X 0,Y 342.747,Z 961.836,A -85,B 0,C 180,E1 21210.014,E2 21210.014} C_VEL
LIN {X 0,Y 343.84,Z 963.709,A -85,B 0,C 180,E1 21210.748,E2 21210.748} C_VEL
LIN {X 0,Y 346.178,Z 971.468,A -85,B 0,C 180,E1 21212.461,E2 21212.461} C_VEL
LIN {X 0,Y 349.708,Z 987.54,A -85,B 0,C 180,E1 21214.951,E2 21214.951} C_VEL
LIN {X 0,Y 355.813,Z 1005.024,A -85,B 0,C 180,E1 21217.697,E2 21217.697} C_VEL
LIN {X 0,Y 351.96,Z 1039.781,A -85,B 0,C 180,E1 21219.518,E2 21219.518} C_VEL
LIN {X 0,Y 346.164,Z 1067.132,A -85,B 0,C 180,E1 21221.882,E2 21221.882} C_VEL
LIN {X 0,Y 339.358,Z 1089.696,A -85,B 0,C 180,E1 21224.838,E2 21224.838} C_VEL
LIN {X 0,Y 331.85,Z 1109.086,A -85,B 0,C 180,E1 21228.702,E2 21228.702} C_VEL
LIN {X 0,Y 325.441,Z 1121.903,A -85,B 0,C 180,E1 21232.667,E2 21232.667} C_VEL
LIN {X 0,Y 319.722,Z 1130.423,A -85,B 0,C 180,E1 21237.294,E2 21237.294} C_VEL
LIN {X 0,Y 317.198,Z 1132.885,A -85,B 0,C 180,E1 21240.003,E2 21240.003} C_VEL
LIN {X 0,Y 315.257,Z 1133.7,A -85,B 0,C 180,E1 21242.75,E2 21242.75} C_VEL
LIN {X 0,Y 313.262,Z 1131.928,A -85,B 0,C 180,E1 21246.805,E2 21246.805} C_VEL
LIN {X 0,Y 312.367,Z 1124.708,A -85,B 0,C 180,E1 21251.867,E2 21251.867} C_VEL
LIN {X 0,Y 312.676,Z 1111.665,A -85,B 0,C 180,E1 21256.859,E2 21256.859} C_VEL
LIN {X 0,Y 313.829,Z 1094.066,A -85,B 0,C 180,E1 21261.173,E2 21261.173} C_VEL
LIN {X 0,Y 315.65,Z 1071.16,A -85,B 0,C 180,E1 21265.023,E2 21265.023} C_VEL
LIN {X 0,Y 317.713,Z 1042.805,A -85,B 0,C 180,E1 21268.209,E2 21268.209} C_VEL
LIN {X 0,Y 319.299,Z 1012.377,A -85,B 0,C 180,E1 21270.334,E2 21270.334} C_VEL
LIN {X 0,Y 319.401,Z 980.111,A -85,B 0,C 180,E1 21271.578,E2 21271.578} C_VEL
LIN {X 0,Y 307.327,Z 923.03,A -85,B 0,C 180,E1 21274.075,E2 21274.075} C_VEL
LIN {X 0,Y 306.817,Z 923.03,A -85,B 0,C 180,E1 21282.343,E2 21282.343} C_VEL
LIN {X 0,Y 306.844,Z 923.03,A -85,B 0,C 180,E1 21290.165,E2 21290.165} C_VEL
LIN {X 0,Y 306.998,Z 923.03,A -85,B 0,C 180,E1 21297.192,E2 21297.192} C_VEL
LIN {X 0,Y 307.405,Z 923.03,A -85,B 0,C 180,E1 21303.717,E2 21303.717} C_VEL
LIN {X 0,Y 307.792,Z 923.03,A -85,B 0,C 180,E1 21309.875,E2 21309.875} C_VEL
LIN {X 0,Y 308.483,Z 923.03,A -85,B 0,C 180,E1 21318.449,E2 21318.449} C_VEL
LIN {X 0,Y 309.425,Z 923.03,A -85,B 0,C 180,E1 21327.176,E2 21327.176} C_VEL
LIN {X 0,Y 309.413,Z 923.03,A -85,B 0,C 180,E1 21332.774,E2 21332.774} C_VEL
LIN {X 0,Y 308.54,Z 923.03,A -85,B 0,C 180,E1 21341.602,E2 21341.602} C_VEL
LIN {X 0,Y 307.824,Z 923.03,A -85,B 0,C 180,E1 21350.07,E2 21350.07} C_VEL
LIN {X 0,Y 307.288,Z 923.03,A -85,B 0,C 180,E1 21357.723,E2 21357.723} C_VEL
LIN {X 0,Y 306.898,Z 923.03,A -85,B 0,C 180,E1 21366.183,E2 21366.183} C_VEL
LIN {X 0,Y 306.942,Z 923.03,A -85,B 0,C 180,E1 21370.479,E2 21370.479} C_VEL
LIN {X 0,Y 324.764,Z 969.823,A -85,B 0,C 180,E1 21374.774,E2 21374.774} C_VEL
LIN {X 0,Y 336.779,Z 1009.46,A -85,B 0,C 180,E1 21378.777,E2 21378.777} C_VEL
LIN {X 0,Y 341.837,Z 1031.872,A -85,B 0,C 180,E1 21381.25,E2 21381.25} C_VEL
LIN {X 0,Y 333.716,Z 1069.741,A -85,B 0,C 180,E1 21385.13,E2 21385.13} C_VEL
LIN {X 0,Y 326.018,Z 1102.37,A -85,B 0,C 180,E1 21389.728,E2 21389.728} C_VEL
LIN {X 0,Y 319.302,Z 1130.733,A -85,B 0,C 180,E1 21395.162,E2 21395.162} C_VEL
LIN {X 0,Y 314.273,Z 1154.404,A -85,B 0,C 180,E1 21401.422,E2 21401.422} C_VEL
LIN {X 0,Y 311.325,Z 1172.149,A -85,B 0,C 180,E1 21408.092,E2 21408.092} C_VEL
LIN {X 0,Y 310.146,Z 1183.357,A -85,B 0,C 180,E1 21414.405,E2 21414.405} C_VEL
LIN {X 0,Y 309.981,Z 1189.282,A -85,B 0,C 180,E1 21419.997,E2 21419.997} C_VEL
LIN {X 0,Y 310.604,Z 1191.911,A -85,B 0,C 180,E1 21425.581,E2 21425.581} C_VEL
LIN {X 0,Y 312.514,Z 1191.286,A -85,B 0,C 180,E1 21431.149,E2 21431.149} C_VEL
LIN {X 0,Y 317.435,Z 1186.153,A -85,B 0,C 180,E1 21438.21,E2 21438.21} C_VEL
LIN {X 0,Y 326.742,Z 1175.433,A -85,B 0,C 180,E1 21445.42,E2 21445.42} C_VEL
LIN {X 0,Y 342.34,Z 1157.701,A -85,B 0,C 180,E1 21452.655,E2 21452.655} C_VEL
LIN {X 0,Y 363.473,Z 1134.12,A -85,B 0,C 180,E1 21458.954,E2 21458.954} C_VEL
LIN {X 0,Y 387.274,Z 1107.976,A -85,B 0,C 180,E1 21463.694,E2 21463.694} C_VEL
LIN {X 0,Y 385.809,Z 1109.815,A -85,B 0,C 180,E1 21464.191,E2 21464.191} C_VEL
LIN {X 0,Y 361.395,Z 1139.452,A -85,B 0,C 180,E1 21468.728,E2 21468.728} C_VEL
LIN {X 0,Y 338.671,Z 1169.301,A -85,B 0,C 180,E1 21475.364,E2 21475.364} C_VEL
LIN {X 0,Y 323.232,Z 1191.902,A -85,B 0,C 180,E1 21482.801,E2 21482.801} C_VEL
LIN {X 0,Y 314.542,Z 1207.107,A -85,B 0,C 180,E1 21490.377,E2 21490.377} C_VEL
LIN {X 0,Y 310.835,Z 1215.674,A -85,B 0,C 180,E1 21497.464,E2 21497.464} C_VEL
LIN {X 0,Y 309.919,Z 1219.117,A -85,B 0,C 180,E1 21504.429,E2 21504.429} C_VEL
LIN {X 0,Y 310.294,Z 1217.978,A -85,B 0,C 180,E1 21510.025,E2 21510.025} C_VEL
LIN {X 0,Y 310.4,Z 1213.11,A -85,B 0,C 180,E1 21515.612,E2 21515.612} C_VEL
LIN {X 0,Y 310.87,Z 1202.666,A -85,B 0,C 180,E1 21521.909,E2 21521.909} C_VEL
LIN {X 0,Y 312.965,Z 1186.274,A -85,B 0,C 180,E1 21528.315,E2 21528.315} C_VEL
LIN {X 0,Y 317.43,Z 1163.164,A -85,B 0,C 180,E1 21534.64,E2 21534.64} C_VEL
LIN {X 0,Y 323.994,Z 1134.575,A -85,B 0,C 180,E1 21540.238,E2 21540.238} C_VEL
LIN {X 0,Y 331.783,Z 1101.671,A -85,B 0,C 180,E1 21544.939,E2 21544.939} C_VEL
LIN {X 0,Y 340.176,Z 1063.648,A -85,B 0,C 180,E1 21548.857,E2 21548.857} C_VEL
LIN {X 0,Y 346.177,Z 1030.358,A -85,B 0,C 180,E1 21551.33,E2 21551.33} C_VEL
LIN {X 0,Y 332.763,Z 988.465,A -85,B 0,C 180,E1 21555.141,E2 21555.141} C_VEL
LIN {X 0,Y 331.666,Z 983.653,A -85,B 0,C 180,E1 21555.791,E2 21555.791} C_VEL
LIN {X 0,Y 334.531,Z 959.975,A -85,B 0,C 180,E1 21559.6,E2 21559.6} C_VEL
LIN {X 0,Y 336.299,Z 961.329,A -85,B 0,C 180,E1 21565.652,E2 21565.652} C_VEL
LIN {X 0,Y 340.578,Z 969.572,A -85,B 0,C 180,E1 21569.853,E2 21569.853} C_VEL
LIN {X 0,Y 346.412,Z 980.427,A -85,B 0,C 180,E1 21573.344,E2 21573.344} C_VEL
LIN {X 0,Y 349.708,Z 987.54,A -85,B 0,C 180,E1 21574.951,E2 21574.951} C_VEL
LIN {X 0,Y 351.427,Z 996.027,A -85,B 0,C 180,E1 21576.03,E2 21576.03} C_VEL
LIN {X 0,Y 351.051,Z 1010.836,A -85,B 0,C 180,E1 21576.916,E2 21576.916} C_VEL
LIN {X 0,Y 350.164,Z 1019.672,A -85,B 0,C 180,E1 21577.307,E2 21577.307} C_VEL
LIN {X 0,Y 345.284,Z 1049.709,A -85,B 0,C 180,E1 21579.174,E2 21579.174} C_VEL
LIN {X 0,Y 339.01,Z 1074.818,A -85,B 0,C 180,E1 21581.654,E2 21581.654} C_VEL
LIN {X 0,Y 331.637,Z 1096.168,A -85,B 0,C 180,E1 21584.814,E2 21584.814} C_VEL
LIN {X 0,Y 324.069,Z 1113.442,A -85,B 0,C 180,E1 21588.672,E2 21588.672} C_VEL
LIN {X 0,Y 316.931,Z 1125.979,A -85,B 0,C 180,E1 21593.157,E2 21593.157} C_VEL
LIN {X 0,Y 310.926,Z 1133.206,A -85,B 0,C 180,E1 21598.2,E2 21598.2} C_VEL
LIN {X 0,Y 307.333,Z 1134.764,A -85,B 0,C 180,E1 21602.821,E2 21602.821} C_VEL
LIN {X 0,Y 305.089,Z 1131.64,A -85,B 0,C 180,E1 21607.719,E2 21607.719} C_VEL
LIN {X 0,Y 304.43,Z 1122.886,A -85,B 0,C 180,E1 21612.91,E2 21612.91} C_VEL
LIN {X 0,Y 304.977,Z 1108.196,A -85,B 0,C 180,E1 21617.96,E2 21617.96} C_VEL
LIN {X 0,Y 306.487,Z 1088.121,A -85,B 0,C 180,E1 21622.467,E2 21622.467} C_VEL
LIN {X 0,Y 308.453,Z 1063.74,A -85,B 0,C 180,E1 21626.165,E2 21626.165} C_VEL
LIN {X 0,Y 310.334,Z 1035.29,A -85,B 0,C 180,E1 21629.047,E2 21629.047} C_VEL
LIN {X 0,Y 311.874,Z 1003.003,A -85,B 0,C 180,E1 21630.99,E2 21630.99} C_VEL
LIN {X 0,Y 311.481,Z 980.461,A -85,B 0,C 180,E1 21631.807,E2 21631.807} C_VEL
LIN {X 0,Y 299.38,Z 923.03,A -85,B 0,C 180,E1 21634.256,E2 21634.256} C_VEL
LIN {X 0,Y 298.861,Z 923.03,A -85,B 0,C 180,E1 21641.099,E2 21641.099} C_VEL
LIN {X 0,Y 298.877,Z 923.03,A -85,B 0,C 180,E1 21649.327,E2 21649.327} C_VEL
LIN {X 0,Y 298.992,Z 923.03,A -85,B 0,C 180,E1 21656.198,E2 21656.198} C_VEL
LIN {X 0,Y 299.449,Z 923.03,A -85,B 0,C 180,E1 21662.963,E2 21662.963} C_VEL
LIN {X 0,Y 299.825,Z 923.03,A -85,B 0,C 180,E1 21669.316,E2 21669.316} C_VEL
LIN {X 0,Y 300.282,Z 923.03,A -85,B 0,C 180,E1 21675.402,E2 21675.402} C_VEL
LIN {X 0,Y 300.798,Z 923.03,A -85,B 0,C 180,E1 21681.307,E2 21681.307} C_VEL
LIN {X 0,Y 301.81,Z 923.03,A -85,B 0,C 180,E1 21689.975,E2 21689.975} C_VEL
LIN {X 0,Y 300.875,Z 923.03,A -85,B 0,C 180,E1 21698.639,E2 21698.639} C_VEL
LIN {X 0,Y 300.2,Z 923.03,A -85,B 0,C 180,E1 21706.972,E2 21706.972} C_VEL
LIN {X 0,Y 299.517,Z 923.03,A -85,B 0,C 180,E1 21714.746,E2 21714.746} C_VEL
LIN {X 0,Y 299.141,Z 923.03,A -85,B 0,C 180,E1 21720.818,E2 21720.818} C_VEL
LIN {X 0,Y 298.986,Z 923.03,A -85,B 0,C 180,E1 21729.537,E2 21729.537} C_VEL
LIN {X 0,Y 317.243,Z 970.91,A -85,B 0,C 180,E1 21734.12,E2 21734.12} C_VEL
LIN {X 0,Y 329.117,Z 1010.129,A -85,B 0,C 180,E1 21738.213,E2 21738.213} C_VEL
LIN {X 0,Y 334.257,Z 1033.645,A -85,B 0,C 180,E1 21740.872,E2 21740.872} C_VEL
LIN {X 0,Y 326,Z 1071.029,A -85,B 0,C 180,E1 21744.816,E2 21744.816} C_VEL
LIN {X 0,Y 317.973,Z 1104.354,A -85,B 0,C 180,E1 21749.67,E2 21749.67} C_VEL
LIN {X 0,Y 310.905,Z 1133.8,A -85,B 0,C 180,E1 21755.595,E2 21755.595} C_VEL
LIN {X 0,Y 305.981,Z 1156.751,A -85,B 0,C 180,E1 21762.018,E2 21762.018} C_VEL
LIN {X 0,Y 303.299,Z 1173.168,A -85,B 0,C 180,E1 21768.502,E2 21768.502} C_VEL
LIN {X 0,Y 302.266,Z 1183.234,A -85,B 0,C 180,E1 21774.259,E2 21774.259} C_VEL
LIN {X 0,Y 302.077,Z 1189.907,A -85,B 0,C 180,E1 21780.641,E2 21780.641} C_VEL
LIN {X 0,Y 303.622,Z 1192.561,A -85,B 0,C 180,E1 21788.584,E2 21788.584} C_VEL
LIN {X 0,Y 307.355,Z 1189.846,A -85,B 0,C 180,E1 21795.685,E2 21795.685} C_VEL
LIN {X 0,Y 316.506,Z 1180.711,A -85,B 0,C 180,E1 21803.939,E2 21803.939} C_VEL
LIN {X 0,Y 331.553,Z 1165.102,A -85,B 0,C 180,E1 21811.606,E2 21811.606} C_VEL
LIN {X 0,Y 352.88,Z 1143.37,A -85,B 0,C 180,E1 21818.38,E2 21818.38} C_VEL
LIN {X 0,Y 378.108,Z 1117.9,A -85,B 0,C 180,E1 21823.626,E2 21823.626} C_VEL
LIN {X 0,Y 376.253,Z 1120.039,A -85,B 0,C 180,E1 21824.154,E2 21824.154} C_VEL
LIN {X 0,Y 348.169,Z 1151.905,A -85,B 0,C 180,E1 21829.823,E2 21829.823} C_VEL
LIN {X 0,Y 327.746,Z 1177.182,A -85,B 0,C 180,E1 21836.44,E2 21836.44} C_VEL
LIN {X 0,Y 313.014,Z 1197.499,A -85,B 0,C 180,E1 21844.277,E2 21844.277} C_VEL
LIN {X 0,Y 305.881,Z 1209.374,A -85,B 0,C 180,E1 21851.298,E2 21851.298} C_VEL
LIN {X 0,Y 302.652,Z 1216.544,A -85,B 0,C 180,E1 21858.507,E2 21858.507} C_VEL
LIN {X 0,Y 302.025,Z 1218.614,A -85,B 0,C 180,E1 21864.283,E2 21864.283} C_VEL
LIN {X 0,Y 302.43,Z 1217.274,A -85,B 0,C 180,E1 21870.025,E2 21870.025} C_VEL
LIN {X 0,Y 302.526,Z 1212.16,A -85,B 0,C 180,E1 21875.758,E2 21875.758} C_VEL
LIN {X 0,Y 303.049,Z 1201.558,A -85,B 0,C 180,E1 21882.146,E2 21882.146} C_VEL
LIN {X 0,Y 305.252,Z 1184.621,A -85,B 0,C 180,E1 21888.795,E2 21888.795} C_VEL
LIN {X 0,Y 310.071,Z 1160.896,A -85,B 0,C 180,E1 21895.265,E2 21895.265} C_VEL
LIN {X 0,Y 316.586,Z 1132.934,A -85,B 0,C 180,E1 21900.784,E2 21900.784} C_VEL
LIN {X 0,Y 324.745,Z 1099.257,A -85,B 0,C 180,E1 21905.632,E2 21905.632} C_VEL
LIN {X 0,Y 333.51,Z 1060.234,A -85,B 0,C 180,E1 21909.628,E2 21909.628} C_VEL
LIN {X 0,Y 338.676,Z 1031.865,A -85,B 0,C 180,E1 21911.773,E2 21911.773} C_VEL
LIN {X 0,Y 328.887,Z 999.553,A -85,B 0,C 180,E1 21915.002,E2 21915.002} C_VEL
LIN {X 0,Y 332.61,Z 967.663,A -85,B 0,C 180,E1 21920.137,E2 21920.137} C_VEL
LIN {X 0,Y 334.349,Z 969.285,A -85,B 0,C 180,E1 21925.56,E2 21925.56} C_VEL
LIN {X 0,Y 338.34,Z 977.104,A -85,B 0,C 180,E1 21929.632,E2 21929.632} C_VEL
LIN {X 0,Y 344.268,Z 989.204,A -85,B 0,C 180,E1 21933.357,E2 21933.357} C_VEL
LIN {X 0,Y 350.14,Z 1005.013,A -85,B 0,C 180,E1 21936.303,E2 21936.303} C_VEL
LIN {X 0,Y 351.177,Z 1009.977,A -85,B 0,C 180,E1 21936.895,E2 21936.895} C_VEL
LIN {X 0,Y 350.164,Z 1019.672,A -85,B 0,C 180,E1 21937.307,E2 21937.307} C_VEL
LIN {X 0,Y 345.52,Z 1036.494,A -85,B 0,C 180,E1 21937.682,E2 21937.682} C_VEL
LIN {X 0,Y 340.594,Z 1050.729,A -85,B 0,C 180,E1 21938.137,E2 21938.137} C_VEL
LIN {X 0,Y 340.141,Z 1052.643,A -85,B 0,C 180,E1 21938.275,E2 21938.275} C_VEL
LIN {X 0,Y 332.952,Z 1078.59,A -85,B 0,C 180,E1 21940.964,E2 21940.964} C_VEL
LIN {X 0,Y 324.57,Z 1100.728,A -85,B 0,C 180,E1 21944.475,E2 21944.475} C_VEL
LIN {X 0,Y 315.723,Z 1118.617,A -85,B 0,C 180,E1 21948.966,E2 21948.966} C_VEL
LIN {X 0,Y 308.379,Z 1129.626,A -85,B 0,C 180,E1 21953.673,E2 21953.673} C_VEL
LIN {X 0,Y 302.376,Z 1135.325,A -85,B 0,C 180,E1 21958.941,E2 21958.941} C_VEL
LIN {X 0,Y 299.42,Z 1135.755,A -85,B 0,C 180,E1 21962.896,E2 21962.896} C_VEL
LIN {X 0,Y 297.248,Z 1132.283,A -85,B 0,C 180,E1 21967.624,E2 21967.624} C_VEL
LIN {X 0,Y 296.55,Z 1122.811,A -85,B 0,C 180,E1 21973.111,E2 21973.111} C_VEL
LIN {X 0,Y 297.108,Z 1108.063,A -85,B 0,C 180,E1 21978.09,E2 21978.09} C_VEL
LIN {X 0,Y 298.673,Z 1087.541,A -85,B 0,C 180,E1 21982.695,E2 21982.695} C_VEL
LIN {X 0,Y 300.76,Z 1061.817,A -85,B 0,C 180,E1 21986.586,E2 21986.586} C_VEL
LIN {X 0,Y 302.756,Z 1032.343,A -85,B 0,C 180,E1 21989.491,E2 21989.491} C_VEL
LIN {X 0,Y 304.147,Z 1000.632,A -85,B 0,C 180,E1 21991.313,E2 21991.313} C_VEL
LIN {X 0,Y 303.532,Z 980.526,A -85,B 0,C 180,E1 21992.053,E2 21992.053} C_VEL
LIN {X 0,Y 291.396,Z 923.03,A -85,B 0,C 180,E1 21994.681,E2 21994.681} C_VEL
LIN {X 0,Y 290.773,Z 923.03,A -85,B 0,C 180,E1 22003.286,E2 22003.286} C_VEL
LIN {X 0,Y 290.867,Z 923.03,A -85,B 0,C 180,E1 22011.405,E2 22011.405} C_VEL
LIN {X 0,Y 291.167,Z 923.03,A -85,B 0,C 180,E1 22018.709,E2 22018.709} C_VEL
LIN {X 0,Y 291.63,Z 923.03,A -85,B 0,C 180,E1 22025.484,E2 22025.484} C_VEL
LIN {X 0,Y 292.047,Z 923.03,A -85,B 0,C 180,E1 22031.888,E2 22031.888} C_VEL
LIN {X 0,Y 292.665,Z 923.03,A -85,B 0,C 180,E1 22038.834,E2 22038.834} C_VEL
LIN {X 0,Y 293.572,Z 923.03,A -85,B 0,C 180,E1 22047.024,E2 22047.024} C_VEL
LIN {X 0,Y 293.561,Z 923.03,A -85,B 0,C 180,E1 22052.924,E2 22052.924} C_VEL
LIN {X 0,Y 292.695,Z 923.03,A -85,B 0,C 180,E1 22061.89,E2 22061.89} C_VEL
LIN {X 0,Y 292.097,Z 923.03,A -85,B 0,C 180,E1 22068.054,E2 22068.054} C_VEL
LIN {X 0,Y 291.634,Z 923.03,A -85,B 0,C 180,E1 22074.458,E2 22074.458} C_VEL
LIN {X 0,Y 291.208,Z 923.03,A -85,B 0,C 180,E1 22081.225,E2 22081.225} C_VEL
LIN {X 0,Y 291.03,Z 923.03,A -85,B 0,C 180,E1 22088.622,E2 22088.622} C_VEL
LIN {X 0,Y 309.137,Z 970.212,A -85,B 0,C 180,E1 22093.28,E2 22093.28} C_VEL
LIN {X 0,Y 321.217,Z 1009.807,A -85,B 0,C 180,E1 22097.519,E2 22097.519} C_VEL
LIN {X 0,Y 326.674,Z 1035.307,A -85,B 0,C 180,E1 22100.484,E2 22100.484} C_VEL
LIN {X 0,Y 318.518,Z 1071.284,A -85,B 0,C 180,E1 22104.369,E2 22104.369} C_VEL
LIN {X 0,Y 310.429,Z 1104.231,A -85,B 0,C 180,E1 22109.258,E2 22109.258} C_VEL
LIN {X 0,Y 303.171,Z 1133.832,A -85,B 0,C 180,E1 22115.324,E2 22115.324} C_VEL
LIN {X 0,Y 298.328,Z 1155.813,A -85,B 0,C 180,E1 22121.541,E2 22121.541} C_VEL
LIN {X 0,Y 295.477,Z 1172.659,A -85,B 0,C 180,E1 22128.193,E2 22128.193} C_VEL
LIN {X 0,Y 294.38,Z 1182.994,A -85,B 0,C 180,E1 22134.104,E2 22134.104} C_VEL
LIN {X 0,Y 294.236,Z 1189.54,A -85,B 0,C 180,E1 22139.997,E2 22139.997} C_VEL
LIN {X 0,Y 294.88,Z 1192.679,A -85,B 0,C 180,E1 22145.879,E2 22145.879} C_VEL
LIN {X 0,Y 297.014,Z 1192.743,A -85,B 0,C 180,E1 22151.739,E2 22151.739} C_VEL
LIN {X 0,Y 303.922,Z 1187.361,A -85,B 0,C 180,E1 22160.364,E2 22160.364} C_VEL
LIN {X 0,Y 316.508,Z 1175.688,A -85,B 0,C 180,E1 22168.514,E2 22168.514} C_VEL
LIN {X 0,Y 335.828,Z 1157.709,A -85,B 0,C 180,E1 22175.957,E2 22175.957} C_VEL
LIN {X 0,Y 361.963,Z 1133.453,A -85,B 0,C 180,E1 22182.309,E2 22182.309} C_VEL
LIN {X 0,Y 368.097,Z 1127.862,A -85,B 0,C 180,E1 22183.438,E2 22183.438} C_VEL
LIN {X 0,Y 368.503,Z 1127.559,A -85,B 0,C 180,E1 22183.84,E2 22183.84} C_VEL
LIN {X 0,Y 340.489,Z 1157.05,A -85,B 0,C 180,E1 22189.563,E2 22189.563} C_VEL
LIN {X 0,Y 319.8,Z 1180.697,A -85,B 0,C 180,E1 22196.308,E2 22196.308} C_VEL
LIN {X 0,Y 304.912,Z 1199.577,A -85,B 0,C 180,E1 22204.332,E2 22204.332} C_VEL
LIN {X 0,Y 297.276,Z 1211.304,A -85,B 0,C 180,E1 22212.271,E2 22212.271} C_VEL
LIN {X 0,Y 294.82,Z 1216.275,A -85,B 0,C 180,E1 22218.197,E2 22218.197} C_VEL
LIN {X 0,Y 294.13,Z 1218.106,A -85,B 0,C 180,E1 22224.129,E2 22224.129} C_VEL
LIN {X 0,Y 294.569,Z 1216.555,A -85,B 0,C 180,E1 22230.026,E2 22230.026} C_VEL
LIN {X 0,Y 294.675,Z 1211.107,A -85,B 0,C 180,E1 22235.912,E2 22235.912} C_VEL
LIN {X 0,Y 295.294,Z 1199.53,A -85,B 0,C 180,E1 22242.793,E2 22242.793} C_VEL
LIN {X 0,Y 297.816,Z 1181.768,A -85,B 0,C 180,E1 22249.625,E2 22249.625} C_VEL
LIN {X 0,Y 302.645,Z 1158.705,A -85,B 0,C 180,E1 22255.893,E2 22255.893} C_VEL
LIN {X 0,Y 309.53,Z 1130.03,A -85,B 0,C 180,E1 22261.565,E2 22261.565} C_VEL
LIN {X 0,Y 318.04,Z 1095.629,A -85,B 0,C 180,E1 22266.486,E2 22266.486} C_VEL
LIN {X 0,Y 326.758,Z 1057.292,A -85,B 0,C 180,E1 22270.374,E2 22270.374} C_VEL
LIN {X 0,Y 331.293,Z 1033.806,A -85,B 0,C 180,E1 22272.171,E2 22272.171} C_VEL
LIN {X 0,Y 326.203,Z 1015.897,A -85,B 0,C 180,E1 22274.111,E2 22274.111} C_VEL
LIN {X 0,Y 330.763,Z 975.428,A -85,B 0,C 180,E1 22280.753,E2 22280.753} C_VEL
LIN {X 0,Y 332.402,Z 976.998,A -85,B 0,C 180,E1 22285.399,E2 22285.399} C_VEL
LIN {X 0,Y 336.192,Z 984.815,A -85,B 0,C 180,E1 22289.481,E2 22289.481} C_VEL
LIN {X 0,Y 341.719,Z 997.074,A -85,B 0,C 180,E1 22293.142,E2 22293.142} C_VEL
LIN {X 0,Y 346.678,Z 1012.086,A -85,B 0,C 180,E1 22295.86,E2 22295.86} C_VEL
LIN {X 0,Y 342.372,Z 1042.326,A -85,B 0,C 180,E1 22297.489,E2 22297.489} C_VEL
LIN {X 0,Y 340.141,Z 1052.643,A -85,B 0,C 180,E1 22298.275,E2 22298.275} C_VEL
LIN {X 0,Y 333.991,Z 1068.323,A -85,B 0,C 180,E1 22299.138,E2 22299.138} C_VEL
LIN {X 0,Y 327.541,Z 1081.116,A -85,B 0,C 180,E1 22300.08,E2 22300.08} C_VEL
LIN {X 0,Y 326.852,Z 1082.796,A -85,B 0,C 180,E1 22300.293,E2 22300.293} C_VEL
LIN {X 0,Y 317.501,Z 1105.13,A -85,B 0,C 180,E1 22304.121,E2 22304.121} C_VEL
LIN {X 0,Y 308.304,Z 1121.758,A -85,B 0,C 180,E1 22308.697,E2 22308.697} C_VEL
LIN {X 0,Y 300.704,Z 1131.927,A -85,B 0,C 180,E1 22313.511,E2 22313.511} C_VEL
LIN {X 0,Y 296.295,Z 1135.813,A -85,B 0,C 180,E1 22317.08,E2 22317.08} C_VEL
LIN {X 0,Y 293.618,Z 1137.053,A -85,B 0,C 180,E1 22320.003,E2 22320.003} C_VEL
LIN {X 0,Y 290.614,Z 1135.814,A -85,B 0,C 180,E1 22324.477,E2 22324.477} C_VEL
LIN {X 0,Y 288.86,Z 1129.601,A -85,B 0,C 180,E1 22329.792,E2 22329.792} C_VEL
LIN {X 0,Y 288.773,Z 1117.766,A -85,B 0,C 180,E1 22335.171,E2 22335.171} C_VEL
LIN {X 0,Y 289.793,Z 1099.91,A -85,B 0,C 180,E1 22340.244,E2 22340.244} C_VEL
LIN {X 0,Y 291.647,Z 1077.77,A -85,B 0,C 180,E1 22344.491,E2 22344.491} C_VEL
LIN {X 0,Y 293.704,Z 1050.691,A -85,B 0,C 180,E1 22348.02,E2 22348.02} C_VEL
LIN {X 0,Y 295.656,Z 1018.857,A -85,B 0,C 180,E1 22350.629,E2 22350.629} C_VEL
LIN {X 0,Y 296.181,Z 983.836,A -85,B 0,C 180,E1 22352.171,E2 22352.171} C_VEL
LIN {X 0,Y 283.411,Z 923.03,A -85,B 0,C 180,E1 22354.991,E2 22354.991} C_VEL
LIN {X 0,Y 282.788,Z 923.03,A -85,B 0,C 180,E1 22364.005,E2 22364.005} C_VEL
LIN {X 0,Y 282.823,Z 923.03,A -85,B 0,C 180,E1 22370.092,E2 22370.092} C_VEL
LIN {X 0,Y 283.254,Z 923.03,A -85,B 0,C 180,E1 22378.608,E2 22378.608} C_VEL
LIN {X 0,Y 283.643,Z 923.03,A -85,B 0,C 180,E1 22384.921,E2 22384.921} C_VEL
LIN {X 0,Y 284.194,Z 923.03,A -85,B 0,C 180,E1 22393.165,E2 22393.165} C_VEL
LIN {X 0,Y 284.901,Z 923.03,A -85,B 0,C 180,E1 22400.818,E2 22400.818} C_VEL
LIN {X 0,Y 285.657,Z 923.03,A -85,B 0,C 180,E1 22406.941,E2 22406.941} C_VEL
LIN {X 0,Y 285.647,Z 923.03,A -85,B 0,C 180,E1 22413.005,E2 22413.005} C_VEL
LIN {X 0,Y 284.716,Z 923.03,A -85,B 0,C 180,E1 22422.228,E2 22422.228} C_VEL
LIN {X 0,Y 284.112,Z 923.03,A -85,B 0,C 180,E1 22428.58,E2 22428.58} C_VEL
LIN {X 0,Y 283.599,Z 923.03,A -85,B 0,C 180,E1 22435.198,E2 22435.198} C_VEL
LIN {X 0,Y 283.22,Z 923.03,A -85,B 0,C 180,E1 22442.21,E2 22442.21} C_VEL
LIN {X 0,Y 283.032,Z 923.03,A -85,B 0,C 180,E1 22447.63,E2 22447.63} C_VEL
LIN {X 0,Y 301.03,Z 969.719,A -85,B 0,C 180,E1 22452.419,E2 22452.419} C_VEL
LIN {X 0,Y 313.361,Z 1009.929,A -85,B 0,C 180,E1 22456.845,E2 22456.845} C_VEL
LIN {X 0,Y 319.308,Z 1035.911,A -85,B 0,C 180,E1 22459.983,E2 22459.983} C_VEL
LIN {X 0,Y 310.823,Z 1072.322,A -85,B 0,C 180,E1 22464.015,E2 22464.015} C_VEL
LIN {X 0,Y 302.257,Z 1106.356,A -85,B 0,C 180,E1 22469.233,E2 22469.233} C_VEL
LIN {X 0,Y 295.007,Z 1135.258,A -85,B 0,C 180,E1 22475.403,E2 22475.403} C_VEL
LIN {X 0,Y 290.217,Z 1156.989,A -85,B 0,C 180,E1 22481.792,E2 22481.792} C_VEL
LIN {X 0,Y 287.474,Z 1173.62,A -85,B 0,C 180,E1 22488.628,E2 22488.628} C_VEL
LIN {X 0,Y 286.407,Z 1184.799,A -85,B 0,C 180,E1 22495.458,E2 22495.458} C_VEL
LIN {X 0,Y 286.351,Z 1190.743,A -85,B 0,C 180,E1 22501.509,E2 22501.509} C_VEL
LIN {X 0,Y 287.973,Z 1193.601,A -85,B 0,C 180,E1 22509.054,E2 22509.054} C_VEL
LIN {X 0,Y 293.466,Z 1190.931,A -85,B 0,C 180,E1 22517.992,E2 22517.992} C_VEL
LIN {X 0,Y 304.698,Z 1182.055,A -85,B 0,C 180,E1 22526.506,E2 22526.506} C_VEL
LIN {X 0,Y 322.253,Z 1167.219,A -85,B 0,C 180,E1 22534.239,E2 22534.239} C_VEL
LIN {X 0,Y 346.341,Z 1146.868,A -85,B 0,C 180,E1 22540.875,E2 22540.875} C_VEL
LIN {X 0,Y 358.014,Z 1137.061,A -85,B 0,C 180,E1 22543.232,E2 22543.232} C_VEL
LIN {X 0,Y 359.298,Z 1136.027,A -85,B 0,C 180,E1 22543.77,E2 22543.77} C_VEL
LIN {X 0,Y 331.726,Z 1162.914,A -85,B 0,C 180,E1 22549.559,E2 22549.559} C_VEL
LIN {X 0,Y 310.277,Z 1185.624,A -85,B 0,C 180,E1 22556.81,E2 22556.81} C_VEL
LIN {X 0,Y 295.904,Z 1202.686,A -85,B 0,C 180,E1 22565.114,E2 22565.114} C_VEL
LIN {X 0,Y 288.76,Z 1212.849,A -85,B 0,C 180,E1 22573.302,E2 22573.302} C_VEL
LIN {X 0,Y 286.439,Z 1217.213,A -85,B 0,C 180,E1 22580.922,E2 22580.922} C_VEL
LIN {X 0,Y 286.42,Z 1217.15,A -85,B 0,C 180,E1 22587.003,E2 22587.003} C_VEL
LIN {X 0,Y 286.77,Z 1213.412,A -85,B 0,C 180,E1 22593.047,E2 22593.047} C_VEL
LIN {X 0,Y 287.055,Z 1204.413,A -85,B 0,C 180,E1 22599.877,E2 22599.877} C_VEL
LIN {X 0,Y 288.766,Z 1188.581,A -85,B 0,C 180,E1 22607.145,E2 22607.145} C_VEL
LIN {X 0,Y 292.946,Z 1166.774,A -85,B 0,C 180,E1 22613.993,E2 22613.993} C_VEL
LIN {X 0,Y 299.386,Z 1143.839,A -85,B 0,C 180,E1 22619.922,E2 22619.922} C_VEL
LIN {X 0,Y 307.397,Z 1116.33,A -85,B 0,C 180,E1 22624.879,E2 22624.879} C_VEL
LIN {X 0,Y 315.228,Z 1085.517,A -85,B 0,C 180,E1 22628.761,E2 22628.761} C_VEL
LIN {X 0,Y 321.628,Z 1051.382,A -85,B 0,C 180,E1 22631.708,E2 22631.708} C_VEL
LIN {X 0,Y 323.805,Z 1034.923,A -85,B 0,C 180,E1 22632.75,E2 22632.75} C_VEL
LIN {X 0,Y 326.655,Z 993.961,A -85,B 0,C 180,E1 22639.592,E2 22639.592} C_VEL
LIN {X 0,Y 328.997,Z 983.001,A -85,B 0,C 180,E1 22641.366,E2 22641.366} C_VEL
LIN {X 0,Y 330.465,Z 984.781,A -85,B 0,C 180,E1 22645.267,E2 22645.267} C_VEL
LIN {X 0,Y 334.137,Z 992.65,A -85,B 0,C 180,E1 22649.384,E2 22649.384} C_VEL
LIN {X 0,Y 339.546,Z 1005.936,A -85,B 0,C 180,E1 22653.148,E2 22653.148} C_VEL
LIN {X 0,Y 342.285,Z 1016.237,A -85,B 0,C 180,E1 22654.898,E2 22654.898} C_VEL
LIN {X 0,Y 337.401,Z 1045.902,A -85,B 0,C 180,E1 22656.582,E2 22656.582} C_VEL
LIN {X 0,Y 330.325,Z 1072.774,A -85,B 0,C 180,E1 22659.063,E2 22659.063} C_VEL
LIN {X 0,Y 326.852,Z 1082.796,A -85,B 0,C 180,E1 22660.293,E2 22660.293} C_VEL
LIN {X 0,Y 319.102,Z 1096.347,A -85,B 0,C 180,E1 22661.757,E2 22661.757} C_VEL
LIN {X 0,Y 311.753,Z 1106.992,A -85,B 0,C 180,E1 22663.22,E2 22663.22} C_VEL
LIN {X 0,Y 310.988,Z 1108.297,A -85,B 0,C 180,E1 22663.502,E2 22663.502} C_VEL
LIN {X 0,Y 301.863,Z 1123.456,A -85,B 0,C 180,E1 22667.87,E2 22667.87} C_VEL
LIN {X 0,Y 294.007,Z 1133.143,A -85,B 0,C 180,E1 22672.621,E2 22672.621} C_VEL
LIN {X 0,Y 287.368,Z 1137.926,A -85,B 0,C 180,E1 22678.128,E2 22678.128} C_VEL
LIN {X 0,Y 282.67,Z 1136.415,A -85,B 0,C 180,E1 22684.603,E2 22684.603} C_VEL
LIN {X 0,Y 280.938,Z 1129.487,A -85,B 0,C 180,E1 22690.071,E2 22690.071} C_VEL
LIN {X 0,Y 280.928,Z 1116.662,A -85,B 0,C 180,E1 22695.605,E2 22695.605} C_VEL
LIN {X 0,Y 281.951,Z 1099.294,A -85,B 0,C 180,E1 22700.485,E2 22700.485} C_VEL
LIN {X 0,Y 283.855,Z 1076.756,A -85,B 0,C 180,E1 22704.789,E2 22704.789} C_VEL
LIN {X 0,Y 285.875,Z 1050.688,A -85,B 0,C 180,E1 22708.195,E2 22708.195} C_VEL
LIN {X 0,Y 287.779,Z 1020.589,A -85,B 0,C 180,E1 22710.726,E2 22710.726} C_VEL
LIN {X 0,Y 288.419,Z 984.968,A -85,B 0,C 180,E1 22712.361,E2 22712.361} C_VEL
LIN {X 0,Y 275.438,Z 923.03,A -85,B 0,C 180,E1 22715.304,E2 22715.304} C_VEL
LIN {X 0,Y 274.882,Z 923.03,A -85,B 0,C 180,E1 22724.352,E2 22724.352} C_VEL
LIN {X 0,Y 274.937,Z 923.03,A -85,B 0,C 180,E1 22732.771,E2 22732.771} C_VEL
LIN {X 0,Y 275.476,Z 923.03,A -85,B 0,C 180,E1 22741.369,E2 22741.369} C_VEL
LIN {X 0,Y 275.902,Z 923.03,A -85,B 0,C 180,E1 22748.613,E2 22748.613} C_VEL
LIN {X 0,Y 276.692,Z 923.03,A -85,B 0,C 180,E1 22757.355,E2 22757.355} C_VEL
LIN {X 0,Y 277.725,Z 923.03,A -85,B 0,C 180,E1 22766.854,E2 22766.854} C_VEL
LIN {X 0,Y 277.716,Z 923.03,A -85,B 0,C 180,E1 22773.091,E2 22773.091} C_VEL
LIN {X 0,Y 276.745,Z 923.03,A -85,B 0,C 180,E1 22782.586,E2 22782.586} C_VEL
LIN {X 0,Y 275.936,Z 923.03,A -85,B 0,C 180,E1 22791.405,E2 22791.405} C_VEL
LIN {X 0,Y 275.403,Z 923.03,A -85,B 0,C 180,E1 22799.557,E2 22799.557} C_VEL
LIN {X 0,Y 275.136,Z 923.03,A -85,B 0,C 180,E1 22806.605,E2 22806.605} C_VEL
LIN {X 0,Y 293.086,Z 969.435,A -85,B 0,C 180,E1 22811.552,E2 22811.552} C_VEL
LIN {X 0,Y 305.191,Z 1008.704,A -85,B 0,C 180,E1 22816.002,E2 22816.002} C_VEL
LIN {X 0,Y 311.722,Z 1037.411,A -85,B 0,C 180,E1 22819.556,E2 22819.556} C_VEL
LIN {X 0,Y 302.722,Z 1074.969,A -85,B 0,C 180,E1 22823.864,E2 22823.864} C_VEL
LIN {X 0,Y 294.318,Z 1107.766,A -85,B 0,C 180,E1 22829.104,E2 22829.104} C_VEL
LIN {X 0,Y 287.252,Z 1135.161,A -85,B 0,C 180,E1 22835.109,E2 22835.109} C_VEL
LIN {X 0,Y 282.36,Z 1157.047,A -85,B 0,C 180,E1 22841.671,E2 22841.671} C_VEL
LIN {X 0,Y 279.659,Z 1173.039,A -85,B 0,C 180,E1 22848.306,E2 22848.306} C_VEL
LIN {X 0,Y 278.53,Z 1184.614,A -85,B 0,C 180,E1 22855.329,E2 22855.329} C_VEL
LIN {X 0,Y 278.644,Z 1191.939,A -85,B 0,C 180,E1 22863.105,E2 22863.105} C_VEL
LIN {X 0,Y 280.155,Z 1194.123,A -85,B 0,C 180,E1 22869.309,E2 22869.309} C_VEL
LIN {X 0,Y 285.995,Z 1191.958,A -85,B 0,C 180,E1 22878.479,E2 22878.479} C_VEL
LIN {X 0,Y 297.811,Z 1183.783,A -85,B 0,C 180,E1 22887.168,E2 22887.168} C_VEL
LIN {X 0,Y 318.014,Z 1168.468,A -85,B 0,C 180,E1 22895.593,E2 22895.593} C_VEL
LIN {X 0,Y 343.433,Z 1148.905,A -85,B 0,C 180,E1 22902.14,E2 22902.14} C_VEL
LIN {X 0,Y 348.25,Z 1145.245,A -85,B 0,C 180,E1 22903.107,E2 22903.107} C_VEL
LIN {X 0,Y 349.909,Z 1144.007,A -85,B 0,C 180,E1 22903.703,E2 22903.703} C_VEL
LIN {X 0,Y 321.848,Z 1169.38,A -85,B 0,C 180,E1 22909.827,E2 22909.827} C_VEL
LIN {X 0,Y 300.786,Z 1190.07,A -85,B 0,C 180,E1 22917.346,E2 22917.346} C_VEL
LIN {X 0,Y 286.906,Z 1205.319,A -85,B 0,C 180,E1 22925.941,E2 22925.941} C_VEL
LIN {X 0,Y 280.306,Z 1213.964,A -85,B 0,C 180,E1 22934.393,E2 22934.393} C_VEL
LIN {X 0,Y 278.561,Z 1216.829,A -85,B 0,C 180,E1 22940.663,E2 22940.663} C_VEL
LIN {X 0,Y 278.555,Z 1216.459,A -85,B 0,C 180,E1 22946.918,E2 22946.918} C_VEL
LIN {X 0,Y 278.919,Z 1212.427,A -85,B 0,C 180,E1 22953.133,E2 22953.133} C_VEL
LIN {X 0,Y 279.155,Z 1204.404,A -85,B 0,C 180,E1 22959.373,E2 22959.373} C_VEL
LIN {X 0,Y 280.772,Z 1188.91,A -85,B 0,C 180,E1 22966.842,E2 22966.842} C_VEL
LIN {X 0,Y 289.231,Z 1155.963,A -85,B 0,C 180,E1 22978.075,E2 22978.075} C_VEL
LIN {X 0,Y 297.489,Z 1131.685,A -85,B 0,C 180,E1 22983.58,E2 22983.58} C_VEL
LIN {X 0,Y 306.957,Z 1101.945,A -85,B 0,C 180,E1 22988.226,E2 22988.226} C_VEL
LIN {X 0,Y 315.439,Z 1069.33,A -85,B 0,C 180,E1 22991.713,E2 22991.713} C_VEL
LIN {X 0,Y 320.974,Z 1038.822,A -85,B 0,C 180,E1 22993.959,E2 22993.959} C_VEL
LIN {X 0,Y 326.522,Z 993.683,A -85,B 0,C 180,E1 23001.529,E2 23001.529} C_VEL
LIN {X 0,Y 327.336,Z 990.679,A -85,B 0,C 180,E1 23002.099,E2 23002.099} C_VEL
LIN {X 0,Y 328.509,Z 992.485,A -85,B 0,C 180,E1 23005.102,E2 23005.102} C_VEL
